   REGION Sequence Next Step Condition
       IF #sCheck_Step_Condition THEN
           CASE #sCurrent_Step_NB OF
               #S00_INIT:
                   REGION S00 INIT
                       IF #sInterface.SequenceReleased AND #iJobReq THEN
                           #sCurrent_Step_NB := #S10_CHECK_INT_LOAD_UNLOAD_OPTION;
                           #sInterface.SequenceRun := TRUE;
                           #sCheck_Step_Condition := FALSE;
                       ELSE
                           #sInterface.SequenceRun := FALSE;
                       END_IF;
                   END_REGION
               #S10_CHECK_INT_LOAD_UNLOAD_OPTION:
                   REGION S10_CHECK_INT_LOAD_UNLOAD_OPTION
                       IF #sInterface.SequenceReleased AND #sStepForward AND "DB_LoaderOptions".IntLoadUnload.CommonPos AND (#iDrilledPartToUnload OR #iUnDrilledPartToLoad) THEN
                           #sCurrent_Step_NB := #S20_SHUTTLE_TO_INT_LOAD_UNLOAD_POS_START_REQ;
                           #sCheck_Step_Condition := FALSE;
                       ELSIF #sInterface.SequenceReleased AND #sStepForward AND "DB_LoaderOptions".IntLoadUnload.CommonPos AND NOT #iJobReq OR (NOT #iDrilledPartToUnload AND NOT #iUnDrilledPartToLoad) THEN
                           #sCurrent_Step_NB := #S260_NO_PART_TO_LOAD_UNLOAD;
                           #sCheck_Step_Condition := FALSE;
                       END_IF;
                   END_REGION
               #S20_SHUTTLE_TO_INT_LOAD_UNLOAD_POS_START_REQ:
                   REGION S20_SHUTTLE_TO_INT_LOAD_UNLOAD_POS_START_REQ
                       IF #sInterface.SequenceReleased AND (#iShuttleMoving OR #iShuttleIntLoadUnloadPos) THEN
                           #sCurrent_Step_NB := #S30_SHUTTLE_TO_INT_LOAD_UNLOAD_POS_REACHED;
                           #sCheck_Step_Condition := FALSE;
                       END_IF;
                   END_REGION
               #S30_SHUTTLE_TO_INT_LOAD_UNLOAD_POS_REACHED:
                   REGION S30_SHUTTLE_TO_INT_LOAD_UNLOAD_POS_REACHED
                       IF #sInterface.SequenceReleased AND #sStepForward AND NOT #sShuttleStartReq AND #iShuttleIntLoadUnloadPos THEN
                           #sCurrent_Step_NB := #S60_AXIS_V_TO_INT_LOAD_UNLOAD_POS_START_REQ;
                           #sCheck_Step_Condition := FALSE;
                       END_IF;
                   END_REGION
               #S40_AXIS_W_TO_SAFE_POS_START_REQ:
                   REGION S40_AXIS_W_TO_SAFE_POS_START_REQ
                       IF #sInterface.SequenceReleased AND #sStepForward AND (#iAxisW_Moving OR #iAxisW_SafePos) THEN
                           #sCurrent_Step_NB := #S50_AXIS_W_TO_SAFE_POS_REACHED;
                           #sCheck_Step_Condition := FALSE;
                       END_IF;
                   END_REGION
               #S50_AXIS_W_TO_SAFE_POS_REACHED:
                   REGION S50_AXIS_W_TO_SAFE_POS_REACHED
                       IF #sInterface.SequenceReleased AND #sStepForward AND NOT #sAxisW_StartReq AND #iAxisW_SafePos THEN
                           #sCurrent_Step_NB := #S60_AXIS_V_TO_INT_LOAD_UNLOAD_POS_START_REQ;
                           #sCheck_Step_Condition := FALSE;
                       END_IF;
                   END_REGION
               #S60_AXIS_V_TO_INT_LOAD_UNLOAD_POS_START_REQ:
                   REGION S60_AXIS_V_TO_INT_LOAD_UNLOAD_POS_START_REQ
                       IF #sInterface.SequenceReleased AND (#iAxisV_Moving OR #iAxisV_LoadUnloadShuttlePos) THEN
                           #sCurrent_Step_NB := #S70_AXIS_V_TO_INT_LOAD_UNLOAD_POS_REACHED;
                           #sCheck_Step_Condition := FALSE;
                       END_IF;
                   END_REGION
               #S70_AXIS_V_TO_INT_LOAD_UNLOAD_POS_REACHED:
                   REGION S70_AXIS_V_TO_INT_LOAD_UNLOAD_POS_REACHED
                       IF #sInterface.SequenceReleased AND #sStepForward AND NOT #sAxisV_StartReq AND #iAxisV_LoadUnloadShuttlePos THEN
                           #sCurrent_Step_NB := #S80_AXIS_W_TO_INT_LOAD_UNLOAD_APPROACH_POS_START_REQ;
                           #sCheck_Step_Condition := FALSE;
                       END_IF;
                   END_REGION
               #S80_AXIS_W_TO_INT_LOAD_UNLOAD_APPROACH_POS_START_REQ:
                   REGION S80_AXIS_W_TO_INT_LOAD_UNLOAD_APPROACH_POS_START_REQ
                       IF #sInterface.SequenceReleased AND (#iAxisW_Moving OR #iAxisW_ApproachLoadUnloadPos) THEN
                           #sCurrent_Step_NB := #S90_AXIS_W_TO_INT_LOAD_UNLOAD_APPROACH_POS_REACHED;
                           #sCheck_Step_Condition := FALSE;
                       END_IF;
                   END_REGION
               #S90_AXIS_W_TO_INT_LOAD_UNLOAD_APPROACH_POS_REACHED:
                   REGION S90_AXIS_W_TO_INT_LOAD_UNLOAD_APPROACH_POS_REACHED
                       IF #sInterface.SequenceReleased AND #sStepForward AND NOT #sAxisW_StartReq AND #iAxisW_ApproachLoadUnloadPos THEN
                           #sCurrent_Step_NB := #S100_AXIS_W_TO_INT_LOAD_UNLOAD_POS_START_REQ;
                           #sCheck_Step_Condition := FALSE;
                       END_IF;
                   END_REGION
               #S100_AXIS_W_TO_INT_LOAD_UNLOAD_POS_START_REQ:
                   REGION S100_AXIS_W_TO_INT_LOAD_UNLOAD_POS_START_REQ
                       IF #sInterface.SequenceReleased AND (#iAxisW_Moving OR #iAxisW_LoadUnloadPos) THEN
                           #sCurrent_Step_NB := #S110_AXIS_W_TO_INT_LOAD_UNLOAD_POS_REACHED;
                           #sCheck_Step_Condition := FALSE;
                       END_IF;
                   END_REGION
               #S110_AXIS_W_TO_INT_LOAD_UNLOAD_POS_REACHED:
                   REGION S110_AXIS_W_TO_INT_LOAD_UNLOAD_POS_REACHED
                       IF #sInterface.SequenceReleased AND #sStepForward AND NOT #sAxisW_StartReq AND #iAxisW_LoadUnloadPos THEN
                           #sCurrent_Step_NB := #S120_CLOSE_LOAD_GRIPPER;
                           #sCheck_Step_Condition := FALSE;
                       END_IF;
                   END_REGION
               #S120_CLOSE_LOAD_GRIPPER:
                   REGION S120_CLOSE_LOAD_GRIPPER
                       IF #sInterface.SequenceReleased AND #sStepForward
                           AND ((#iUnDrilledPartToLoad AND #iLoadGripperClosed) OR NOT #iUnDrilledPartToLoad) THEN
                           #sCurrent_Step_NB := #S130_AXIS_W_TO_SAFE_POS_START_REQ;
                           #sCheck_Step_Condition := FALSE;
                       END_IF;
                   END_REGION
               #S130_AXIS_W_TO_SAFE_POS_START_REQ:
                   REGION S130_AXIS_W_TO_SAFE_POS_START_REQ
                       IF #sInterface.SequenceReleased AND (#iAxisW_Moving OR #iAxisW_SafePos) THEN
                           #sCurrent_Step_NB := #S140_AXIS_W_TO_SAFE_POS_REACHED;
                           #sCheck_Step_Condition := FALSE;
                       END_IF;
                   END_REGION
               #S140_AXIS_W_TO_SAFE_POS_REACHED:
                   REGION S140_AXIS_W_TO_SAFE_POS_REACHED
                       IF #sInterface.SequenceReleased AND #sStepForward AND NOT #sAxisW_StartReq AND #iAxisW_SafePos THEN
                           #sCurrent_Step_NB := #S150_SHUTTLE_TO_INT_LOAD_UNLOAD_OP_POS_START_REQ;
                           #sCheck_Step_Condition := FALSE;
                       END_IF;
                   END_REGION
               #S150_SHUTTLE_TO_INT_LOAD_UNLOAD_OP_POS_START_REQ:
                   REGION S150_SHUTTLE_TO_INT_LOAD_UNLOAD_OP_POS_START_REQ
                       IF #sInterface.SequenceReleased AND (#iShuttleMoving OR #iShuttleIntLoadUnloadOP_Pos) THEN
                           #sCurrent_Step_NB := #S160_SHUTTLE_TO_INT_LOAD_UNLOAD_OP_POS_REACHED;
                           #sCheck_Step_Condition := FALSE;
                       END_IF;
                   END_REGION
               #S160_SHUTTLE_TO_INT_LOAD_UNLOAD_OP_POS_REACHED:
                   REGION S160_SHUTTLE_TO_INT_LOAD_UNLOAD_OP_POS_REACHED
                       IF #sInterface.SequenceReleased AND #sStepForward AND NOT #sShuttleStartReq AND #iShuttleIntLoadUnloadOP_Pos THEN
                           #sCurrent_Step_NB := #S170_AXIS_W_TO_INT_LOAD_UNLOAD_APPROACH_POS_START_REQ;
                           #sCheck_Step_Condition := FALSE;
                       END_IF;
                   END_REGION
               #S170_AXIS_W_TO_INT_LOAD_UNLOAD_APPROACH_POS_START_REQ:
                   REGION S170_AXIS_W_TO_INT_LOAD_UNLOAD_APPROACH_POS_START_REQ
                       IF #sInterface.SequenceReleased AND (#iAxisW_Moving OR #iAxisW_ApproachLoadUnloadPos) THEN
                           #sCurrent_Step_NB := #S180_AXIS_W_TO_INT_LOAD_UNLOAD_APPROACH_POS_REACHED;
                           #sCheck_Step_Condition := FALSE;
                       END_IF;
                   END_REGION
               #S180_AXIS_W_TO_INT_LOAD_UNLOAD_APPROACH_POS_REACHED:
                   REGION S180_AXIS_W_TO_INT_LOAD_UNLOAD_APPROACH_POS_REACHED
                       IF #sInterface.SequenceReleased AND #sStepForward AND NOT #sAxisW_StartReq AND #iAxisW_ApproachLoadUnloadPos THEN
                           #sCurrent_Step_NB := #S190_AXIS_W_TO_INT_LOAD_UNLOAD_POS_START_REQ;
                           #sCheck_Step_Condition := FALSE;
                       END_IF;
                   END_REGION
               #S190_AXIS_W_TO_INT_LOAD_UNLOAD_POS_START_REQ:
                   REGION S190_AXIS_W_TO_INT_LOAD_UNLOAD_POS_START_REQ
                       IF #sInterface.SequenceReleased AND (#iAxisW_Moving OR #iAxisW_LoadUnloadPos) THEN
                           #sCurrent_Step_NB := #S200_AXIS_W_TO_INT_LOAD_UNLOAD_POS_REACHED;
                           #sCheck_Step_Condition := FALSE;
                       END_IF;
                   END_REGION
               #S200_AXIS_W_TO_INT_LOAD_UNLOAD_POS_REACHED:
                   REGION S200_AXIS_W_TO_INT_LOAD_UNLOAD_POS_REACHED
                       IF #sInterface.SequenceReleased AND #sStepForward AND NOT #sAxisW_StartReq AND #iAxisW_LoadUnloadPos THEN
                           #sCurrent_Step_NB := #S210_OPEN_UNLOAD_GRIPPER;
                           #sCheck_Step_Condition := FALSE;
                       END_IF;
                   END_REGION
               #S210_OPEN_UNLOAD_GRIPPER:
                   REGION S210_OPEN_UNLOAD_GRIPPER
                       IF #sInterface.SequenceReleased AND #sStepForward
                           AND (#iDrilledPartToUnload AND #iUnloadGripperOpen OR NOT #iDrilledPartToUnload) THEN
                           #sCurrent_Step_NB := #S220_AXIS_W_TO_SAFE_POS_START_REQ;
                           #sCheck_Step_Condition := FALSE;
                       END_IF;
                   END_REGION
               #S220_AXIS_W_TO_SAFE_POS_START_REQ:
                   REGION S220_AXIS_W_TO_SAFE_POS_START_REQ
                       IF #sInterface.SequenceReleased AND (#iAxisW_Moving OR #iAxisW_SafePos) THEN
                           #sCurrent_Step_NB := #S230_AXIS_W_TO_SAFE_POS_REACHED;
                           #sCheck_Step_Condition := FALSE;
                       END_IF;
                   END_REGION
               #S230_AXIS_W_TO_SAFE_POS_REACHED:
                   REGION S230_AXIS_W_TO_SAFE_POS_REACHED
                       IF #sInterface.SequenceReleased AND #sStepForward AND NOT #sAxisW_StartReq AND #iAxisW_SafePos THEN
                           #sCurrent_Step_NB := #S295_JOB_DONE;
                           #sCheck_Step_Condition := FALSE;
                       END_IF;
                   END_REGION
               #S240_AXIS_V_TO_SAFE_POS_START_REQ:
                   REGION S240_AXIS_V_TO_SAFE_POS_START_REQ
                       IF #sInterface.SequenceReleased AND (#iAxisV_Moving OR #iAxisV_SafePos) THEN
                           #sCurrent_Step_NB := #S250_AXIS_V_TO_SAFE_POS_REACHED;
                           #sCheck_Step_Condition := FALSE;
                       END_IF;
                   END_REGION
               #S250_AXIS_V_TO_SAFE_POS_REACHED:
                   REGION S160_AXIS_V_TO_SAFE_POS_REACHED
                       IF #sInterface.SequenceReleased AND #sStepForward AND NOT #sAxisV_StartReq AND #iAxisV_SafePos THEN
                           #sCurrent_Step_NB := #S295_JOB_DONE;
                           #sCheck_Step_Condition := FALSE;
                       END_IF;
                   END_REGION
               #S260_NO_PART_TO_LOAD_UNLOAD:
                   REGION S260_NO_PART_TO_LOAD_UNLOAD
                       IF #sInterface.SequenceReleased AND #sStepForward AND "AlwaysTRUE" THEN
                           #sCurrent_Step_NB := #S220_AXIS_W_TO_SAFE_POS_START_REQ;
                           #sCheck_Step_Condition := FALSE;
                       END_IF;
                   END_REGION
               #S295_JOB_DONE:
                   REGION S95_JOB_DONE
                       IF NOT #iJobReq THEN
                           #sCurrent_Step_NB := #S00_INIT;
                           #sCheck_Step_Condition := FALSE;
                           #sInterface.JobDone := FALSE;
                       END_IF;
                   END_REGION
               ELSE
                   #sInterface.Error := TRUE;
           END_CASE;
       END_IF;
   END_REGION

   REGION Outputs Update
       #oShuttleStartReq := #sShuttleStartReq;
       #oShuttlePosSetPoint := #sShuttlePosSetPoint;
       #oAxisV_StartReq := #sAxisV_StartReq;
       #oAxisV_PosSetPoint := #sAxisV_PosSetPoint;
       #oAxisW_StartReq := #sAxisW_StartReq;
       #oAxisW_PosSetPoint := #sAxisW_PosSetPoint;
       #oLoadGripperCloseReq := #sLoadGripperCloseReq;
       #oUnloadGripperOpenReq := #sUnloadGripperOpenReq;

   END_REGION

   REGION Steps - Date and Time History
       IF #sHistory.Activation THEN
           IF #sHistory.Steps[0] <> #sCurrent_Step_NB THEN
               FOR #tIndex := 98 TO 0 BY -1 DO
                   #sHistory.Steps[#tIndex + 1] := #sHistory.Steps[#tIndex];
                   #sHistory.Date_Time[#tIndex + 1] := #sHistory.Date_Time[#tIndex];
               END_FOR;
               #sHistory.Steps[0] := #sCurrent_Step_NB;
               #sHistory.Date_Time[0] := #iPLC_DateAndTime;
           END_IF;
       END_IF;
   END_REGION

   REGION Steps Text
       #StepText(iErrorCode := #sCurrent_Step_NB,
                 oErrorText => #StepText.oErrorText);
   END_REGION
END_FUNCTION_BLOCK

FUNCTION_BLOCK "FB_PartControl"   // FB58, SCL
{ S7_Optimized_Access := 'TRUE' }
// stored: MemoryReserve 100, SetENOAutomatically false
   VAR_INPUT
      iStartSeqCond : Bool;   // Start Sequence Conditions
      iJobReq : Bool;   // Job Request - From Main
      iCtrlEnabled : Bool;   // Part Control Enable - Param or Condition
      iShuttleCtrlUndrilledPos : Bool;   // Undrilled Pos. Reached (Option Individual Ctrl) - Param
      iShuttleCtrlUndrilledPosSetPoint : LReal;   // Undrilled Pos. Setpoint (Option Individual Ctrl) - Param
      iShuttleCtrlDrilledPos : Bool;   // Drilled Pos. Reached (Option Individual Ctrl) - Param
      iShuttleCtrlDrilledPosSetPoint : LReal;   // Drilled Pos. Setpoint (Option Individual Ctrl) - Param
      iShuttleCtrlPos : Bool;   // Control Pos. Reached (Option Common Ctrl) - Param
      iShuttleCtrlPosSetPoint : LReal;   // Control Pos. Setpoint (Option Common Ctrl) - Param
      iExpectedCtrlUndrilled : Bool;   // Expected result Undrilled Pos.
      iExpectedCtrlDrilled : Bool;   // Expected result Drilled Pos.
      iPartMeasureValue : Real;   // Part Measure Value (Option Analog Measure) - From AI
      iPartMeasureTolMin : Real;   // Part Tol Min Value (Option Analog Measure) - Param
      iPartMeasureTolMax : Real;   // Part Tol Max Value (Option Analog Measure) - Param
      iUndrilledPartPresence : Bool;
      iDrilledPartPresence : Bool;
      iShuttleMoving : Bool;   // Shuttle is moving - From FB_LoaderAxis
      iShuttleInPos : Bool;   // Shuttle pos. reached - From FB_LoaderAxis
      iPLC_DateAndTime : DTL;
      iStepPause : Bool;
   END_VAR
   VAR_OUTPUT
      oShuttleStartReq { ExternalAccessible := 'False'; ExternalVisible := 'False'; ExternalWritable := 'False'} : Bool;   // Shuttle Start Order - To FB_LoaderAxis
      oShuttlePosSetPoint { ExternalAccessible := 'False'; ExternalVisible := 'False'; ExternalWritable := 'False'} : Real;   // Shuttle Position Setpoint - To FB_LoaderAxis
      oPartControlOK : Bool;   // Part OK - To Main
      oPartControlNOK : Bool;   // Part NOK - To Main
   END_VAR
   VAR
      sCurrent_Step_NB : Int;   // Active Step Number
      sCheck_Step_Condition : Bool;
      sOneStepForward : Bool;
      sRTOneStepForward : R_TRIG;
      sOneStepMode { S7_SetPoint := 'True'} : Bool;
      sStepForward : Bool;
      sInterface : "UDT_SequenceInterface";
      sShuttleStartReq { ExternalAccessible := 'False'; ExternalVisible := 'False'; ExternalWritable := 'False'} : Bool;
      sShuttlePosSetPoint { ExternalAccessible := 'False'; ExternalVisible := 'False'; ExternalWritable := 'False'} : Real;
      sMissingPartCtrlUndrilled : Bool;
      sMissingPartCtrlDrilled : Bool;
      sExtraPartCtrlUndrilled : Bool;
      sExtraPartCtrlDrilled : Bool;
      sPresencePartUndrilledPos : Bool;
      sPresencePartDrilledPos : Bool;
      sPartControlOK : Bool;
      sPartControlNOK : Bool;
      sControlTimer : TON_TIME;
      sHistory : Struct
         Activation : Bool;
         Steps : Array[0..99] of Int;
         Date_Time : Array[0..99] of DTL;
      END_STRUCT;
      StepText : "FB_GetTextErrorCode";
   END_VAR
   VAR_TEMP
      tIndex : Int;   // Index
   END_VAR
   VAR CONSTANT
      S00_INIT : Int := 0;
      S10_CHECK_PART_PRESENCE_OPTION : Int := 10;
      S20_SHUTTLE_TO_UNDRILLED_POS_START_REQ : Int := 20;
      S30_SHUTTLE_TO_UNDRILLED_POS_REACHED : Int := 30;
      S40_WAIT_UNDRILLED_CTRL_EXECUTION : Int := 40;
      S50_SHUTTLE_TO_DRILLED_POS_START_REQ : Int := 50;
      S60_SHUTTLE_TO_DRILLED_POS_REACHED : Int := 60;
      S70_WAIT_DRILLED_CTRL_EXECUTION : Int := 70;
      S80_CHECK_PART_POS_RESULT : Int := 80;
      S120_SHUTTLE_TO_CONTROL_POS_START_REQ : Int := 120;
      S130_SHUTTLE_TO_CONTROL_POS_REACHED : Int := 130;
      S140_WAIT_CONTROL_EXECUTION : Int := 140;
      S180_CHECK_PART_POS_RESULT : Int := 180;
      S280_NO_PART_CTRL : Int := 280;
      S295_JOB_DONE : Int := 295;
   END_VAR
   // StepText.sCode_error[0].ErrorCode := 0;
   // StepText.sCode_error[1].ErrorCode := 10;
   // StepText.sCode_error[2].ErrorCode := 20;
   // StepText.sCode_error[3].ErrorCode := 30;
   // StepText.sCode_error[4].ErrorCode := 40;
   // StepText.sCode_error[5].ErrorCode := 50;
   // StepText.sCode_error[6].ErrorCode := 60;
   // StepText.sCode_error[7].ErrorCode := 70;
   // StepText.sCode_error[8].ErrorCode := 80;
   // StepText.sCode_error[9].ErrorCode := 90;
   // StepText.sCode_error[10].ErrorCode := 95;
BEGIN
   REGION Description header 
       //==================================================================================
       // POSALUX Swiss SA / (C) Copyright 2025
       //----------------------------------------------------------------------------------
       // Title: FB_PartControl
       // Comment/Function: 
       // Author: Fabien WALDT
       // Engineering: TIA Portal v17
       //----------------------------------------------------------------------------------
       // Change log table:
       // Version  | Date     | Expert in charge | Changes applied
       // ---------|----------|------------------|-----------------------------------------
       // 00.00.01 | 20250527 | WFA              | First released version
       // =================================================================================
   END_REGION

   REGION Define condition to start
       IF #iStartSeqCond THEN
           #sInterface.SequenceReleased := TRUE;
       ELSE
           // Standard sequencer controls
           #sInterface.SequenceReleased := FALSE;
           #sCurrent_Step_NB := #S00_INIT;
           #sInterface.SequenceRun := FALSE;
           #sInterface.JobDone := FALSE;
           #sCheck_Step_Condition := FALSE;

           // Dedicated sequencer controls
           #sShuttleStartReq := FALSE;
           #sShuttlePosSetPoint := 0.0;
           #sPresencePartUndrilledPos := FALSE;
           #sPresencePartDrilledPos := FALSE;

           // Add specifics controls 
       END_IF;

       // Reset interface error
       IF #sInterface.Reset THEN
           #sInterface.Error := FALSE;
       END_IF;

       // Reset start when axis in position
       IF #iShuttleInPos THEN
           #sShuttleStartReq := FALSE;
       END_IF;

       // One step forward
       #sRTOneStepForward.CLK := #sOneStepForward;
       #sRTOneStepForward();
       #sStepForward := (NOT #sOneStepMode OR (#sOneStepMode AND #sRTOneStepForward.Q)) AND NOT #iStepPause;
       #sOneStepForward := FALSE;

       // Step Timer
       #sControlTimer(IN := #sCurrent_Step_NB = 40 OR #sCurrent_Step_NB = 140,
                            PT := T#50ms);
   END_REGION

   REGION Sequence Function
       CASE #sCurrent_Step_NB OF
           #S00_INIT:
               REGION S00 INIT
                   #sCheck_Step_Condition := TRUE;
               END_REGION
           #S10_CHECK_PART_PRESENCE_OPTION:
               REGION S10_CHECK_PART_PRESENCE_OPTION
                   #sPartControlOK := FALSE;
                   #sPartControlNOK := FALSE;
                   #sMissingPartCtrlUndrilled := FALSE;
                   #sMissingPartCtrlDrilled := FALSE;
                   #sExtraPartCtrlUndrilled := FALSE;
                   #sExtraPartCtrlDrilled := FALSE;
                   #sCheck_Step_Condition := TRUE;
               END_REGION
           #S20_SHUTTLE_TO_UNDRILLED_POS_START_REQ:
               REGION S20_SHUTTLE_TO_UNDRILLED_POS_START_REQ
                   #sShuttleStartReq := NOT #iShuttleCtrlUndrilledPos;
                   #sShuttlePosSetPoint := LREAL_TO_REAL(#iShuttleCtrlUndrilledPosSetPoint);
                   #sCheck_Step_Condition := TRUE;
               END_REGION
           #S30_SHUTTLE_TO_UNDRILLED_POS_REACHED:
               REGION S30_SHUTTLE_TO_UNDRILLED_POS_REACHED
                   #sCheck_Step_Condition := TRUE;
               END_REGION
           #S40_WAIT_UNDRILLED_CTRL_EXECUTION:
               REGION S40_WAIT_UNDRILLED_CTRL_EXECUTION
                   IF "DB_LoaderOptions".PartControl.AnalogMeasure THEN
                       IF #iPartMeasureValue > #iPartMeasureTolMin AND #iPartMeasureValue < #iPartMeasureTolMax THEN
                           #sPresencePartUndrilledPos := TRUE;
                       ELSE
                           #sPresencePartUndrilledPos := FALSE;
                       END_IF;
                   ELSIF "DB_LoaderOptions".PartControl.DigitalMeasure THEN
                       IF #iUndrilledPartPresence THEN
                           #sPresencePartUndrilledPos := TRUE;
                       ELSE
                           #sPresencePartUndrilledPos := FALSE;
                       END_IF;
                       IF #iDrilledPartPresence THEN
                           #sPresencePartDrilledPos := TRUE;
                       ELSE
                           #sPresencePartDrilledPos := FALSE;
                       END_IF;
                   ELSE
                       #sInterface.Error := TRUE;
                   END_IF;
                   IF #sControlTimer.Q THEN
                       #sCheck_Step_Condition := TRUE;
                   END_IF;
               END_REGION
           #S50_SHUTTLE_TO_DRILLED_POS_START_REQ:
               REGION S50_SHUTTLE_TO_DRILLED_POS_START_REQ
                   #sShuttleStartReq := NOT #iShuttleCtrlDrilledPos;
                   #sShuttlePosSetPoint := LREAL_TO_REAL(#iShuttleCtrlDrilledPosSetPoint);
                   #sCheck_Step_Condition := TRUE;
               END_REGION
           #S60_SHUTTLE_TO_DRILLED_POS_REACHED:
               REGION S60_SHUTTLE_TO_DRILLED_POS_REACHED
                   #sCheck_Step_Condition := TRUE;
               END_REGION
           #S70_WAIT_DRILLED_CTRL_EXECUTION:
               REGION S70_WAIT_DRILLED_CTRL_EXECUTION
                   IF "DB_LoaderOptions".PartControl.AnalogMeasure THEN
                       IF #iPartMeasureValue > #iPartMeasureTolMin AND #iPartMeasureValue < #iPartMeasureTolMax THEN
                           #sPresencePartUndrilledPos := TRUE;
                       ELSE
                           #sPresencePartUndrilledPos := FALSE;
                       END_IF;
                   ELSIF "DB_LoaderOptions".PartControl.DigitalMeasure THEN
                       IF #iUndrilledPartPresence THEN
                           #sPresencePartUndrilledPos := TRUE;
                       ELSE
                           #sPresencePartUndrilledPos := FALSE;
                       END_IF;
                   ELSE
                       #sInterface.Error := TRUE;
                   END_IF;
                   #sCheck_Step_Condition := TRUE;
               END_REGION
           #S80_CHECK_PART_POS_RESULT:
               REGION S80_CHECK_PART_POS_RESULT
                   #sExtraPartCtrlUndrilled := #sPresencePartUndrilledPos AND NOT #iExpectedCtrlUndrilled;
                   #sMissingPartCtrlUndrilled := NOT #sPresencePartUndrilledPos AND #iExpectedCtrlUndrilled;
                   #sExtraPartCtrlDrilled := #sPresencePartDrilledPos AND NOT #iExpectedCtrlDrilled;
                   #sMissingPartCtrlDrilled := NOT #sPresencePartDrilledPos AND #iExpectedCtrlDrilled;

                   IF #sPresencePartUndrilledPos = #iExpectedCtrlUndrilled AND #sPresencePartDrilledPos = #iExpectedCtrlDrilled THEN
                       #sPartControlOK := TRUE;
                       #sPartControlNOK := FALSE;
                   ELSE
                       #sPartControlOK := FALSE;
                       #sPartControlNOK := TRUE;
                   END_IF;
                   #sCheck_Step_Condition := TRUE;
               END_REGION

           #S120_SHUTTLE_TO_CONTROL_POS_START_REQ:
               REGION S120_SHUTTLE_TO_CONTROL_POS_START_REQ
                   #sShuttleStartReq := NOT #iShuttleCtrlPos;
                   #sShuttlePosSetPoint := LREAL_TO_REAL(#iShuttleCtrlPosSetPoint);
                   #sCheck_Step_Condition := TRUE;
               END_REGION
           #S130_SHUTTLE_TO_CONTROL_POS_REACHED:
               REGION S130_SHUTTLE_TO_CONTROL_POS_REACHED
                   #sCheck_Step_Condition := TRUE;
               END_REGION
           #S140_WAIT_CONTROL_EXECUTION:
               REGION S140_WAIT_CONTROL_EXECUTION
                   IF "DB_LoaderOptions".PartControl.AnalogMeasure THEN
                       IF #iPartMeasureValue > #iPartMeasureTolMin AND #iPartMeasureValue < #iPartMeasureTolMax THEN
                           #sPresencePartUndrilledPos := TRUE;
                       ELSE
                           #sPresencePartUndrilledPos := FALSE;
                       END_IF;
                   ELSIF "DB_LoaderOptions".PartControl.DigitalMeasure THEN
                       IF #iUndrilledPartPresence THEN
                           #sPresencePartUndrilledPos := TRUE;
                       ELSE
                           #sPresencePartUndrilledPos := FALSE;
                       END_IF;
                       IF #iDrilledPartPresence THEN
                           #sPresencePartDrilledPos := TRUE;
                       ELSE
                           #sPresencePartDrilledPos := FALSE;
                       END_IF;
                   ELSE
                       #sInterface.Error := TRUE;
                   END_IF;
                   IF #sControlTimer.Q THEN
                       #sCheck_Step_Condition := TRUE;
                   END_IF;
               END_REGION
           #S180_CHECK_PART_POS_RESULT:
               REGION S180_CHECK_PART_POS_RESULT
                   #sExtraPartCtrlUndrilled := #sPresencePartUndrilledPos AND NOT #iExpectedCtrlUndrilled;
                   #sMissingPartCtrlUndrilled := NOT #sPresencePartUndrilledPos AND #iExpectedCtrlUndrilled;
                   #sExtraPartCtrlDrilled := #sPresencePartDrilledPos AND NOT #iExpectedCtrlDrilled;
                   #sMissingPartCtrlDrilled := NOT #sPresencePartDrilledPos AND #iExpectedCtrlDrilled;

                   IF #sPresencePartUndrilledPos = #iExpectedCtrlUndrilled AND #sPresencePartDrilledPos = #iExpectedCtrlDrilled THEN
                       #sPartControlOK := TRUE;
                       #sPartControlNOK := FALSE;
                   ELSE
                       #sPartControlOK := FALSE;
                       #sPartControlNOK := TRUE;
                   END_IF;
                   #sCheck_Step_Condition := TRUE;
               END_REGION

           #S280_NO_PART_CTRL:
               REGION S280_NO_PART_CTRL
                   #sPartControlOK := TRUE;
                   #sPartControlNOK := FALSE;
                   #sCheck_Step_Condition := TRUE;
               END_REGION

           #S295_JOB_DONE:
               REGION S295_JOB_DONE
                   #sInterface.JobDone := TRUE;
                   #sCheck_Step_Condition := TRUE;
               END_REGION
           ELSE:
               #sInterface.Error := TRUE;
       END_CASE;
   END_REGION

   REGION Sequence Next Step Condition
       IF #sCheck_Step_Condition THEN
           CASE #sCurrent_Step_NB OF
               #S00_INIT:
                   REGION S00 INIT
                       IF #sInterface.SequenceReleased AND #iJobReq THEN
                           #sCurrent_Step_NB := #S10_CHECK_PART_PRESENCE_OPTION;
                           #sInterface.SequenceRun := TRUE;
                           #sCheck_Step_Condition := FALSE;
                       ELSE
                           #sInterface.SequenceRun := FALSE;
                       END_IF;
                   END_REGION
               #S10_CHECK_PART_PRESENCE_OPTION:
                   REGION S10_CHECK_PART_PRESENCE_OPTION
                       IF #sInterface.SequenceReleased AND #sStepForward AND "DB_LoaderOptions".PartControl.Individual AND (NOT "DB_LoaderOptions".PartControl.Disabled AND #iCtrlEnabled) THEN
                           #sCurrent_Step_NB := #S20_SHUTTLE_TO_UNDRILLED_POS_START_REQ;
                           #sCheck_Step_Condition := FALSE;
                       ELSIF #sInterface.SequenceReleased AND #sStepForward AND "DB_LoaderOptions".PartControl.Common AND (NOT "DB_LoaderOptions".PartControl.Disabled AND #iCtrlEnabled) THEN
                           #sCurrent_Step_NB := #S120_SHUTTLE_TO_CONTROL_POS_START_REQ;
                           #sCheck_Step_Condition := FALSE;
                       ELSIF #sInterface.SequenceReleased AND #sStepForward AND ("DB_LoaderOptions".PartControl.Disabled OR NOT #iCtrlEnabled) THEN
                           #sCurrent_Step_NB := #S280_NO_PART_CTRL;
                           #sCheck_Step_Condition := FALSE;
                       END_IF;
                   END_REGION
               #S20_SHUTTLE_TO_UNDRILLED_POS_START_REQ:
                   REGION S20_SHUTTLE_TO_UNDRILLED_POS_START_REQ
                       IF #sInterface.SequenceReleased AND (#iShuttleMoving OR #iShuttleCtrlUndrilledPos) THEN
                           #sCurrent_Step_NB := #S30_SHUTTLE_TO_UNDRILLED_POS_REACHED;
                           #sCheck_Step_Condition := FALSE;
                       END_IF;
                   END_REGION
               #S30_SHUTTLE_TO_UNDRILLED_POS_REACHED:
                   REGION S30_SHUTTLE_TO_UNDRILLED_POS_REACHED
                       IF #sInterface.SequenceReleased AND #sStepForward AND NOT #sShuttleStartReq AND #iShuttleCtrlUndrilledPos THEN
                           #sCurrent_Step_NB := #S40_WAIT_UNDRILLED_CTRL_EXECUTION;
                           #sCheck_Step_Condition := FALSE;
                       END_IF;
                   END_REGION
               #S40_WAIT_UNDRILLED_CTRL_EXECUTION:
                   REGION S40_WAIT_UNDRILLED_CTRL_EXECUTION
                       IF #sInterface.SequenceReleased AND #sStepForward AND "AlwaysTRUE" THEN
                           #sCurrent_Step_NB := #S50_SHUTTLE_TO_DRILLED_POS_START_REQ;
                           #sCheck_Step_Condition := FALSE;
                       END_IF;
                   END_REGION
               #S50_SHUTTLE_TO_DRILLED_POS_START_REQ:
                   REGION S50_SHUTTLE_TO_DRILLED_POS_START_REQ
                       IF #sInterface.SequenceReleased AND (#iShuttleMoving OR #iShuttleCtrlDrilledPos) THEN
                           #sCurrent_Step_NB := #S60_SHUTTLE_TO_DRILLED_POS_REACHED;
                           #sCheck_Step_Condition := FALSE;
                       END_IF;
                   END_REGION
               #S60_SHUTTLE_TO_DRILLED_POS_REACHED:
                   REGION S60_SHUTTLE_TO_DRILLED_POS_REACHED
                       IF #sInterface.SequenceReleased AND #sStepForward AND NOT #sShuttleStartReq AND #iShuttleCtrlDrilledPos THEN
                           #sCurrent_Step_NB := #S70_WAIT_DRILLED_CTRL_EXECUTION;
                           #sCheck_Step_Condition := FALSE;
                       END_IF;
                   END_REGION
               #S70_WAIT_DRILLED_CTRL_EXECUTION:
                   REGION S70_WAIT_DRILLED_CTRL_EXECUTION
                       IF #sInterface.SequenceReleased AND #sStepForward AND "AlwaysTRUE" THEN
                           #sCurrent_Step_NB := #S80_CHECK_PART_POS_RESULT;
                           #sCheck_Step_Condition := FALSE;
                       END_IF;
                   END_REGION
               #S80_CHECK_PART_POS_RESULT:
                   REGION S80_CHECK_PART_POS_RESULT
                       IF #sInterface.SequenceReleased AND #sStepForward AND "AlwaysTRUE" THEN
                           #sCurrent_Step_NB := #S295_JOB_DONE;
                           #sCheck_Step_Condition := FALSE;
                       END_IF;
                   END_REGION

               #S120_SHUTTLE_TO_CONTROL_POS_START_REQ:
                   REGION S120_SHUTTLE_TO_CONTROL_POS_START_REQ
                       IF #sInterface.SequenceReleased AND (#iShuttleMoving OR #iShuttleCtrlPos) THEN
                           #sCurrent_Step_NB := #S130_SHUTTLE_TO_CONTROL_POS_REACHED;
                           #sCheck_Step_Condition := FALSE;
                       END_IF;
                   END_REGION
               #S130_SHUTTLE_TO_CONTROL_POS_REACHED:
                   REGION S130_SHUTTLE_TO_CONTROL_POS_REACHED
                       IF #sInterface.SequenceReleased AND #sStepForward AND NOT #sShuttleStartReq AND #iShuttleCtrlPos THEN
                           #sCurrent_Step_NB := #S140_WAIT_CONTROL_EXECUTION;
                           #sCheck_Step_Condition := FALSE;
                       END_IF;
                   END_REGION
               #S140_WAIT_CONTROL_EXECUTION:
                   REGION S140_WAIT_CONTROL_EXECUTION
                       IF #sInterface.SequenceReleased AND #sStepForward AND "AlwaysTRUE" THEN
                           #sCurrent_Step_NB := #S180_CHECK_PART_POS_RESULT;
                           #sCheck_Step_Condition := FALSE;
                       END_IF;
                   END_REGION
               #S180_CHECK_PART_POS_RESULT:
                   REGION S180_CHECK_PART_POS_RESULT
                       IF #sInterface.SequenceReleased AND #sStepForward AND "AlwaysTRUE" THEN
                           #sCurrent_Step_NB := #S295_JOB_DONE;
                           #sCheck_Step_Condition := FALSE;
                       END_IF;
                   END_REGION

               #S280_NO_PART_CTRL:
                   REGION S280_NO_PART_CTRL
                       IF #sInterface.SequenceReleased AND #sStepForward AND "AlwaysTRUE" THEN
                           #sCurrent_Step_NB := #S295_JOB_DONE;
                           #sCheck_Step_Condition := FALSE;
                       END_IF;
                   END_REGION

               #S295_JOB_DONE:
                   REGION S95_JOB_DONE
                       IF NOT #iJobReq THEN
                           #sCurrent_Step_NB := #S00_INIT;
                           #sCheck_Step_Condition := FALSE;
                           #sInterface.JobDone := FALSE;
                       END_IF;
                   END_REGION
               ELSE
                   #sInterface.Error := TRUE;
           END_CASE;
       END_IF;
   END_REGION

   REGION Outputs Update
       #oShuttleStartReq := #sShuttleStartReq;
       #oShuttlePosSetPoint:= #sShuttlePosSetPoint;
       #oPartControlOK := #sPartControlOK;
       #oPartControlNOK := #sPartControlNOK;
   END_REGION

   REGION Steps - Date and Time History
       IF #sHistory.Activation THEN
           IF #sHistory.Steps[0] <> #sCurrent_Step_NB THEN
               FOR #tIndex := 98 TO 0 BY -1 DO
                   #sHistory.Steps[#tIndex + 1] := #sHistory.Steps[#tIndex];
                   #sHistory.Date_Time[#tIndex + 1] := #sHistory.Date_Time[#tIndex];
               END_FOR;
               #sHistory.Steps[0] := #sCurrent_Step_NB;
               #sHistory.Date_Time[0] := #iPLC_DateAndTime;
           END_IF;
       END_IF;
   END_REGION

   REGION Steps Text
       #StepText(iErrorCode := #sCurrent_Step_NB,
                 oErrorText => #StepText.oErrorText);
   END_REGION
END_FUNCTION_BLOCK

FUNCTION_BLOCK "FB_BwLoadUnload"   // FB72, SCL
{ S7_Optimized_Access := 'TRUE' }
// stored: AutoNumber false, MemoryReserve 100, SetENOAutomatically false
   VAR_INPUT
      iStartSeqCond : Bool;   // Start Sequence Conditions
      iJobReq : Bool;   // Job Request - From Main
      iLoadReq : Bool;   // Load Request - From Main
      iUnloadReq : Bool;   // Unload Request - From Main
      iShuttleBwUnloadPos : Bool;   // Unload Pos. Reached - Param
      iShuttleBwUnloadPosSetPoint : LReal;   // Unload Pos. Setpoint - Param
      iShuttleBwLoadPos : Bool;   // Load Pos. Reached - Param
      iShuttleBwLoadPosSetPoint : LReal;   // Load Pos. Setpoint - Param
      iShuttleMoving : Bool;   // Shuttle is moving - From FB_LoaderAxis
      iShuttleInPos : Bool;   // Shuttle pos. reached - From FB_LoaderAxis
      iBwLoadDone : Bool;
      iBwUnloadDone : Bool;
      iBwLoaderInSafePos : Bool;   // Gripper in Safe Position - Param
      iPLC_DateAndTime : DTL;
      iStepPause : Bool;
   END_VAR
   VAR_OUTPUT
      oShuttleStartReq { ExternalAccessible := 'False'; ExternalVisible := 'False'; ExternalWritable := 'False'} : Bool;   // Shuttle Start Order - To FB_LoaderAxis
      oShuttlePosSetPoint { ExternalAccessible := 'False'; ExternalVisible := 'False'; ExternalWritable := 'False'} : Real;   // Shuttle Position Setpoint - To FB_LoaderAxis
      oBwLoadReq : Bool;
      oBwUnloadReq : Bool;
   END_VAR
   VAR
      sCurrent_Step_NB : Int;   // Active Step Number
      sCheck_Step_Condition : Bool;
      sOneStepForward : Bool;
      sRTOneStepForward : R_TRIG;
      sOneStepMode { S7_SetPoint := 'True'} : Bool;
      sStepForward : Bool;
      sInterface : "UDT_SequenceInterface";
      sShuttleStartReq { ExternalAccessible := 'False'; ExternalVisible := 'False'; ExternalWritable := 'False'} : Bool;
      sShuttlePosSetPoint { ExternalAccessible := 'False'; ExternalVisible := 'False'; ExternalWritable := 'False'} : Real;
      sBwLoadReq : Bool;
      sBwUnloadReq : Bool;
      sHistory : Struct
         Activation : Bool;
         Steps : Array[0..99] of Int;
         Date_Time : Array[0..99] of DTL;
      END_STRUCT;
      StepText : "FB_GetTextErrorCode";
   END_VAR
   VAR_TEMP
      tIndex : Int;   // Index
   END_VAR
   VAR CONSTANT
      S00_INIT : Int := 0;
      S10_BW_LOAD_UNLOAD_OPTION : Int := 10;
      S20_SHUTTLE_TO_BW_LOAD_POS_START_REQ : Int := 20;
      S30_SHUTTLE_TO_BW_LOAD_POS_REACHED : Int := 30;
      S40_SET_EXCHANGE_BW_LOADER_LOAD : Int := 40;
      S50_EXCHANGE_BW_LOADER_IN_PROGRESS : Int := 50;
      S60_EXCHANGE_BW_LOADER_ACQUIT : Int := 60;
      S120_SHUTTLE_TO_BW_UNLOAD_POS_START_REQ : Int := 120;
      S130_SHUTTLE_TO_BW_UNLOAD_POS_REACHED : Int := 130;
      S140_SET_EXCHANGE_BW_LOADER_UNLOAD : Int := 140;
      S150_EXCHANGE_BW_LOADER_IN_PROGRESS : Int := 150;
      S160_EXCHANGE_BW_LOADER_ACQUIT : Int := 160;
      S195_JOB_DONE : Int := 195;
   END_VAR
   // StepText.sCode_error[0].ErrorCode := 0;
   // StepText.sCode_error[1].ErrorCode := 10;
   // StepText.sCode_error[2].ErrorCode := 20;
   // StepText.sCode_error[3].ErrorCode := 30;
   // StepText.sCode_error[4].ErrorCode := 40;
   // StepText.sCode_error[5].ErrorCode := 50;
   // StepText.sCode_error[6].ErrorCode := 60;
   // StepText.sCode_error[7].ErrorCode := 70;
   // StepText.sCode_error[8].ErrorCode := 80;
   // StepText.sCode_error[9].ErrorCode := 90;
   // StepText.sCode_error[10].ErrorCode := 95;
BEGIN
   REGION Description header 
       //==================================================================================
       // POSALUX Swiss SA / (C) Copyright 2025
       //----------------------------------------------------------------------------------
       // Title: FB_BWLoadUnload
       // Comment/Function: 
       // Author: Fabien WALDT
       // Engineering: TIA Portal v17
       //----------------------------------------------------------------------------------
       // Change log table:
       // Version  | Date     | Expert in charge | Changes applied
       // ---------|----------|------------------|-----------------------------------------
       // 00.00.01 | 20250527 | WFA              | First released version
       // =================================================================================
   END_REGION

   REGION Define condition to start
       IF #iStartSeqCond THEN
           #sInterface.SequenceReleased := TRUE;
       ELSE
           // Standard sequencer controls
           #sInterface.SequenceReleased := FALSE;
           #sCurrent_Step_NB := #S00_INIT;
           #sInterface.SequenceRun := FALSE;
           #sInterface.JobDone := FALSE;
           #sCheck_Step_Condition := FALSE;

           // Dedicated sequencer controls
           #sShuttleStartReq := FALSE;
           #sShuttlePosSetPoint := 0.0;
           #sBwLoadReq := FALSE;
           #sBwUnloadReq := FALSE;
           // Add specifics controls 
       END_IF;

       // Reset interface error
       IF #sInterface.Reset THEN
           #sInterface.Error := FALSE;
       END_IF;

       // Reset start when axis in position
       IF #iShuttleInPos THEN
           #sShuttleStartReq := FALSE;
       END_IF;

       // One step forward
       #sRTOneStepForward.CLK := #sOneStepForward;
       #sRTOneStepForward();
       #sStepForward := (NOT #sOneStepMode OR (#sOneStepMode AND #sRTOneStepForward.Q)) AND NOT #iStepPause;
       #sOneStepForward := FALSE;

       // Action only true in dedicated steps

   END_REGION

   REGION Sequence Function
       CASE #sCurrent_Step_NB OF
           #S00_INIT:
               REGION S00 INIT
                   #sBwLoadReq := FALSE;
                   #sBwUnloadReq := FALSE;
                   #sCheck_Step_Condition := TRUE;
               END_REGION
           #S10_BW_LOAD_UNLOAD_OPTION:
               REGION S10_BW_LOAD_UNLOAD_OPTION

                   #sCheck_Step_Condition := TRUE;
               END_REGION
           #S20_SHUTTLE_TO_BW_LOAD_POS_START_REQ:
               REGION S20_SHUTTLE_TO_BW_LOAD_POS_START_REQ
                   #sShuttleStartReq := NOT #iShuttleBwLoadPos;
                   #sShuttlePosSetPoint := LREAL_TO_REAL(#iShuttleBwLoadPosSetPoint);
                   #sCheck_Step_Condition := TRUE;
               END_REGION
           #S30_SHUTTLE_TO_BW_LOAD_POS_REACHED:
               REGION S30_SHUTTLE_TO_BW_LOAD_POS_REACHED
                   #sCheck_Step_Condition := TRUE;
               END_REGION
           #S40_SET_EXCHANGE_BW_LOADER_LOAD:
               REGION S40_SET_EXCHANGE_BW_LOADER_LOAD
                   #sBwLoadReq := TRUE;
                   #sCheck_Step_Condition := TRUE;
               END_REGION
           #S50_EXCHANGE_BW_LOADER_IN_PROGRESS:
               REGION S50_EXCHANGE_BW_LOADER_IN_PROGRESS
                   #sCheck_Step_Condition := TRUE;
               END_REGION
           #S60_EXCHANGE_BW_LOADER_ACQUIT:
               REGION S60_EXCHANGE_BW_LOADER_ACQUIT
                   #sBwLoadReq := FALSE;
                   #sCheck_Step_Condition := TRUE;
               END_REGION

           #S120_SHUTTLE_TO_BW_UNLOAD_POS_START_REQ:
               REGION S120_SHUTTLE_TO_BW_UNLOAD_POS_START_REQ
                   #sShuttleStartReq := NOT #iShuttleBwUnloadPos;
                   #sShuttlePosSetPoint := LREAL_TO_REAL(#iShuttleBwUnloadPosSetPoint);
                   #sCheck_Step_Condition := TRUE;
               END_REGION
           #S130_SHUTTLE_TO_BW_UNLOAD_POS_REACHED:
               REGION S130_SHUTTLE_TO_BW_UNLOAD_POS_REACHED
                   #sCheck_Step_Condition := TRUE;
               END_REGION
           #S140_SET_EXCHANGE_BW_LOADER_UNLOAD:
               REGION S140_SET_EXCHANGE_BW_LOADER_UNLOAD
                   #sBwUnloadReq := TRUE;
                   #sCheck_Step_Condition := TRUE;
               END_REGION
           #S150_EXCHANGE_BW_LOADER_IN_PROGRESS:
               REGION S150_EXCHANGE_BW_LOADER_IN_PROGRESS
                   #sCheck_Step_Condition := TRUE;
               END_REGION
           #S160_EXCHANGE_BW_LOADER_ACQUIT:
               REGION S160_EXCHANGE_BW_LOADER_ACQUIT
                   #sBwUnloadReq := FALSE;
                   #sCheck_Step_Condition := TRUE;
               END_REGION
           #S195_JOB_DONE:
               REGION S95_JOB_DONE
                   #sInterface.JobDone := TRUE;
                   #sCheck_Step_Condition := TRUE;
               END_REGION
           ELSE:
               #sInterface.Error := TRUE;
       END_CASE;
   END_REGION

   REGION Sequence Next Step Condition
       IF #sCheck_Step_Condition THEN
           CASE #sCurrent_Step_NB OF
               #S00_INIT:
                   REGION S00 INIT
                       IF #sInterface.SequenceReleased AND #iJobReq THEN
                           #sCurrent_Step_NB := #S10_BW_LOAD_UNLOAD_OPTION;
                           #sInterface.SequenceRun := TRUE;
                           #sCheck_Step_Condition := FALSE;
                       ELSE
                           #sInterface.SequenceRun := FALSE;
                       END_IF;
                   END_REGION
               #S10_BW_LOAD_UNLOAD_OPTION:
                   REGION S10_BW_LOAD_UNLOAD_OPTION
                       IF #sInterface.SequenceReleased AND #sStepForward AND "DB_LoaderOptions".BwLoadUnload.SeparatePos AND #iLoadReq AND NOT #iUnloadReq THEN
                           #sCurrent_Step_NB := #S20_SHUTTLE_TO_BW_LOAD_POS_START_REQ;
                           #sCheck_Step_Condition := FALSE;
                       ELSIF #sInterface.SequenceReleased AND #sStepForward AND "DB_LoaderOptions".BwLoadUnload.SeparatePos AND NOT #iLoadReq AND #iUnloadReq THEN
                           #sCurrent_Step_NB := #S120_SHUTTLE_TO_BW_UNLOAD_POS_START_REQ;
                           #sCheck_Step_Condition := FALSE;
                       ELSIF #sInterface.SequenceReleased AND #sStepForward AND NOT #iLoadReq AND NOT #iUnloadReq THEN
                           #sCurrent_Step_NB := #S195_JOB_DONE;
                           #sCheck_Step_Condition := FALSE;
                       END_IF;
                   END_REGION
               #S20_SHUTTLE_TO_BW_LOAD_POS_START_REQ:
                   REGION S20_SHUTTLE_TO_BW_LOAD_POS_START_REQ
                       IF #sInterface.SequenceReleased AND (#iShuttleMoving OR #iShuttleBwLoadPos) THEN
                           #sCurrent_Step_NB := #S30_SHUTTLE_TO_BW_LOAD_POS_REACHED;
                           #sCheck_Step_Condition := FALSE;
                       END_IF;
                   END_REGION
               #S30_SHUTTLE_TO_BW_LOAD_POS_REACHED:
                   REGION S30_SHUTTLE_TO_BW_LOAD_POS_REACHED
                       IF #sInterface.SequenceReleased AND #sStepForward AND NOT #sShuttleStartReq AND #iShuttleBwLoadPos AND "DB_BwLoaderExchange".Inputs.BwInErrorState = 0 THEN
                           #sCurrent_Step_NB := #S40_SET_EXCHANGE_BW_LOADER_LOAD;
                           #sCheck_Step_Condition := FALSE;
                       END_IF;
                   END_REGION
               #S40_SET_EXCHANGE_BW_LOADER_LOAD:
                   REGION S40_SET_EXCHANGE_BW_LOADER_LOAD
                       IF #sInterface.SequenceReleased AND #sStepForward AND "AlwaysTRUE" THEN
                           #sCurrent_Step_NB := #S50_EXCHANGE_BW_LOADER_IN_PROGRESS;
                           #sCheck_Step_Condition := FALSE;
                       END_IF;
                   END_REGION
               #S50_EXCHANGE_BW_LOADER_IN_PROGRESS:
                   REGION S50_EXCHANGE_BW_LOADER_IN_PROGRESS
                       IF #sInterface.SequenceReleased AND #sStepForward AND (#iBwLoadDone OR "DB_BwLoaderExchange".Inputs.BwInErrorState <> 0) THEN
                           #sCurrent_Step_NB := #S60_EXCHANGE_BW_LOADER_ACQUIT;
                           #sCheck_Step_Condition := FALSE;
                       END_IF;
                   END_REGION
               #S60_EXCHANGE_BW_LOADER_ACQUIT:
                   REGION S60_EXCHANGE_BW_LOADER_ACQUIT
                       IF #sInterface.SequenceReleased AND #sStepForward AND "AlwaysTRUE" THEN
                           #sCurrent_Step_NB := #S195_JOB_DONE;
                           #sCheck_Step_Condition := FALSE;
                       END_IF;
                   END_REGION
               #S120_SHUTTLE_TO_BW_UNLOAD_POS_START_REQ:
                   REGION S120_SHUTTLE_TO_BW_UNLOAD_POS_START_REQ
                       IF #sInterface.SequenceReleased AND (#iShuttleMoving OR #iShuttleBwUnloadPos) THEN
                           #sCurrent_Step_NB := #S130_SHUTTLE_TO_BW_UNLOAD_POS_REACHED;
                           #sCheck_Step_Condition := FALSE;
                       END_IF;
                   END_REGION
               #S130_SHUTTLE_TO_BW_UNLOAD_POS_REACHED:
                   REGION S130_SHUTTLE_TO_BW_UNLOAD_POS_REACHED
                       IF #sInterface.SequenceReleased AND #sStepForward AND NOT #sShuttleStartReq AND #iShuttleBwUnloadPos AND "DB_BwLoaderExchange".Inputs.BwInErrorState = 0 THEN
                           #sCurrent_Step_NB := #S140_SET_EXCHANGE_BW_LOADER_UNLOAD;
                           #sCheck_Step_Condition := FALSE;
                       END_IF;
                   END_REGION
               #S140_SET_EXCHANGE_BW_LOADER_UNLOAD:
                   REGION S140_SET_EXCHANGE_BW_LOADER_UNLOAD
                       IF #sInterface.SequenceReleased AND #sStepForward AND "AlwaysTRUE" THEN
                           #sCurrent_Step_NB := #S150_EXCHANGE_BW_LOADER_IN_PROGRESS;
                           #sCheck_Step_Condition := FALSE;
                       END_IF;
                   END_REGION
               #S150_EXCHANGE_BW_LOADER_IN_PROGRESS:
                   REGION S150_EXCHANGE_BW_LOADER_IN_PROGRESS
                       IF #sInterface.SequenceReleased AND #sStepForward AND (#iBwUnloadDone OR "DB_BwLoaderExchange".Inputs.BwInErrorState <> 0) THEN
                           #sCurrent_Step_NB := #S160_EXCHANGE_BW_LOADER_ACQUIT;
                           #sCheck_Step_Condition := FALSE;
                       END_IF;
                   END_REGION
               #S160_EXCHANGE_BW_LOADER_ACQUIT:
                   REGION S160_EXCHANGE_BW_LOADER_ACQUIT
                       IF #sInterface.SequenceReleased AND #sStepForward AND "AlwaysTRUE" THEN
                           #sCurrent_Step_NB := #S195_JOB_DONE;
                           #sCheck_Step_Condition := FALSE;
                       END_IF;
                   END_REGION
               #S195_JOB_DONE:
                   REGION S95_JOB_DONE
                       IF NOT #iJobReq THEN
                           #sCurrent_Step_NB := #S00_INIT;
                           #sCheck_Step_Condition := FALSE;
                           #sInterface.JobDone := FALSE;
                       END_IF;
                   END_REGION
               ELSE
                   #sInterface.Error := TRUE;
           END_CASE;
       END_IF;
   END_REGION

   REGION Outputs Update
       #oShuttleStartReq := #sShuttleStartReq;
       #oShuttlePosSetPoint := #sShuttlePosSetPoint;
       #oBwLoadReq := #sBwLoadReq;
       #oBwUnloadReq := #sBwUnloadReq;
   END_REGION

   REGION Steps - Date and Time History
       IF #sHistory.Activation THEN
           IF #sHistory.Steps[0] <> #sCurrent_Step_NB THEN
               FOR #tIndex := 98 TO 0 BY -1 DO
                   #sHistory.Steps[#tIndex + 1] := #sHistory.Steps[#tIndex];
                   #sHistory.Date_Time[#tIndex + 1] := #sHistory.Date_Time[#tIndex];
               END_FOR;
               #sHistory.Steps[0] := #sCurrent_Step_NB;
               #sHistory.Date_Time[0] := #iPLC_DateAndTime;
           END_IF;
       END_IF;
   END_REGION

   REGION Steps Text
       #StepText(iErrorCode := #sCurrent_Step_NB,
                 oErrorText => #StepText.oErrorText);
   END_REGION
END_FUNCTION_BLOCK

FUNCTION_BLOCK "FB_BwControl"   // FB39, SCL
{ S7_Optimized_Access := 'TRUE' }
// stored: MemoryReserve 100, SetENOAutomatically false
   VAR_INPUT
      iStartSeqCond : Bool;   // Start Sequence Conditions
      iJobReq : Bool;   // Job Request - From Main
      iCtrlEnabled : Bool;   // Part Control Enable - Param or Condition
      iShuttleCtrlPos : Bool;   // Control Pos. Reached - Param
      iShuttleCtrlPosSetPoint : LReal;   // Control Pos. Setpoint - Param
      iExpectedCtrl : Bool;   // Expected result ctrl
      iBwPresence : Bool;   // Bw Presence - From DI
      iShuttleMoving : Bool;   // Shuttle is moving - From FB_LoaderAxis
      iShuttleInPos : Bool;   // Shuttle pos. reached - From FB_LoaderAxis
      iPLC_DateAndTime : DTL;
      iStepPause : Bool;
   END_VAR
   VAR_OUTPUT
      oShuttleStartReq { ExternalAccessible := 'False'; ExternalVisible := 'False'; ExternalWritable := 'False'} : Bool;   // Shuttle Start Order - To FB_LoaderAxis
      oShuttlePosSetPoint { ExternalAccessible := 'False'; ExternalVisible := 'False'; ExternalWritable := 'False'} : Real;   // Shuttle Position Setpoint - To FB_LoaderAxis
      oBwControlOK : Bool;   // Bw OK - To Main
      oBwControlNOK : Bool;   // Bw NOK - To Main
   END_VAR
   VAR
      sCurrent_Step_NB : Int;   // Active Step Number
      sCheck_Step_Condition : Bool;
      sOneStepForward : Bool;
      sRTOneStepForward : R_TRIG;
      sOneStepMode { S7_SetPoint := 'True'} : Bool;
      sStepForward : Bool;
      sInterface : "UDT_SequenceInterface";
      sShuttleStartReq { ExternalAccessible := 'False'; ExternalVisible := 'False'; ExternalWritable := 'False'} : Bool;
      sShuttlePosSetPoint { ExternalAccessible := 'False'; ExternalVisible := 'False'; ExternalWritable := 'False'} : Real;
      sMissingBwCtrl : Bool;
      sExtraBwCtrl : Bool;
      sPresenceBw : Bool;
      sBwControlOK : Bool;
      sBwControlNOK : Bool;
      sHistory : Struct
         Activation : Bool;
         Steps : Array[0..99] of Int;
         Date_Time : Array[0..99] of DTL;
      END_STRUCT;
      StepText : "FB_GetTextErrorCode";
   END_VAR
   VAR_TEMP
      tIndex : Int;   // Index
   END_VAR
   VAR CONSTANT
      S00_INIT : Int := 0;
      S10_CHECK_BW_PRESENCE_OPTION : Int := 10;
      S20_SHUTTLE_TO_BW_CTRL_POS_START_REQ : Int := 20;
      S30_SHUTTLE_TO_BW_CTRL_POS_REACHED : Int := 30;
      S40_WAIT_BW_CTRL_EXECUTION : Int := 40;
      S50_CHECK_BW_PRES_RESULT : Int := 50;
      S150_SET_BW_PRES_RESULT : Int := 150;
      S195_JOB_DONE : Int := 195;
   END_VAR
   // StepText.sCode_error[0].ErrorCode := 0;
   // StepText.sCode_error[1].ErrorCode := 10;
   // StepText.sCode_error[2].ErrorCode := 20;
   // StepText.sCode_error[3].ErrorCode := 30;
   // StepText.sCode_error[4].ErrorCode := 40;
   // StepText.sCode_error[5].ErrorCode := 50;
   // StepText.sCode_error[6].ErrorCode := 60;
   // StepText.sCode_error[7].ErrorCode := 70;
   // StepText.sCode_error[8].ErrorCode := 80;
   // StepText.sCode_error[9].ErrorCode := 90;
   // StepText.sCode_error[10].ErrorCode := 95;
BEGIN
   REGION Description header 
       //==================================================================================
       // POSALUX Swiss SA / (C) Copyright 2025
       //----------------------------------------------------------------------------------
       // Title: FB_BwControl
       // Comment/Function: 
       // Author: Fabien WALDT
       // Engineering: TIA Portal v17
       //----------------------------------------------------------------------------------
       // Change log table:
       // Version  | Date     | Expert in charge | Changes applied
       // ---------|----------|------------------|-----------------------------------------
       // 00.00.01 | 20250527 | WFA              | First released version
       // =================================================================================
   END_REGION

   REGION Define condition to start
       IF #iStartSeqCond THEN
           #sInterface.SequenceReleased := TRUE;
       ELSE
           // Standard sequencer controls
           #sInterface.SequenceReleased := FALSE;
           #sCurrent_Step_NB := #S00_INIT;
           #sInterface.SequenceRun := FALSE;
           #sInterface.JobDone := FALSE;
           #sCheck_Step_Condition := FALSE;

           // Dedicated sequencer controls
           #sShuttleStartReq := FALSE;
           #sShuttlePosSetPoint := 0.0;
           #sPresenceBw := FALSE;

           // Add specifics controls 
       END_IF;

       // Reset interface error
       IF #sInterface.Reset THEN
           #sInterface.Error := FALSE;
       END_IF;

       // Reset start when axis in position
       IF #iShuttleInPos THEN
           #sShuttleStartReq := FALSE;
       END_IF;

       // One step forward
       #sRTOneStepForward.CLK := #sOneStepForward;
       #sRTOneStepForward();
       #sStepForward := (NOT #sOneStepMode OR (#sOneStepMode AND #sRTOneStepForward.Q)) AND NOT #iStepPause;
       #sOneStepForward := FALSE;
   END_REGION

   REGION Sequence Function
       CASE #sCurrent_Step_NB OF
           #S00_INIT:
               REGION S00 INIT
                   #sCheck_Step_Condition := TRUE;
               END_REGION
           #S10_CHECK_BW_PRESENCE_OPTION:
               REGION S10_CHECK_BW_PRESENCE_OPTION
                   #sBwControlOK := FALSE;
                   #sBwControlNOK := FALSE;
                   #sMissingBwCtrl := FALSE;
                   #sExtraBwCtrl := FALSE;
                   #sCheck_Step_Condition := TRUE;
               END_REGION
           #S20_SHUTTLE_TO_BW_CTRL_POS_START_REQ:
               REGION S20_SHUTTLE_TO_BW_CTRL_POS_START_REQ
                   #sShuttleStartReq := NOT #iShuttleCtrlPos;
                   #sShuttlePosSetPoint := LREAL_TO_REAL(#iShuttleCtrlPosSetPoint);
                   #sCheck_Step_Condition := TRUE;
               END_REGION
           #S30_SHUTTLE_TO_BW_CTRL_POS_REACHED:
               REGION S30_SHUTTLE_TO_BW_CTRL_POS_REACHED
                   #sCheck_Step_Condition := TRUE;
               END_REGION
           #S40_WAIT_BW_CTRL_EXECUTION:
               REGION S40_WAIT_BW_CTRL_EXECUTION
                   #sPresenceBw := #iBwPresence;
                   #sCheck_Step_Condition := TRUE;
               END_REGION
           #S50_CHECK_BW_PRES_RESULT:
               REGION S50_CHECK_BW_PRES_RESULT
                   #sExtraBwCtrl := #sPresenceBw AND NOT #iExpectedCtrl;
                   #sMissingBwCtrl := NOT #sPresenceBw AND #iExpectedCtrl;
                   IF #sPresenceBw = #iExpectedCtrl THEN
                       #sBwControlOK := TRUE;
                       #sBwControlNOK := FALSE;
                   ELSE
                       #sBwControlOK := FALSE;
                       #sBwControlNOK := TRUE;
                   END_IF;
                   #sCheck_Step_Condition := TRUE;
               END_REGION
           #S150_SET_BW_PRES_RESULT:
               REGION S150_SET_BW_PRES_RESULT
                   #sBwControlOK := TRUE;
                   #sBwControlNOK := FALSE;
                   #sCheck_Step_Condition := TRUE;
               END_REGION
           #S195_JOB_DONE:
               REGION S195_JOB_DONE
                   #sInterface.JobDone := TRUE;
                   #sCheck_Step_Condition := TRUE;
               END_REGION
           ELSE:
               #sInterface.Error := TRUE;
       END_CASE;
   END_REGION

   REGION Sequence Next Step Condition
       IF #sCheck_Step_Condition THEN
           CASE #sCurrent_Step_NB OF
               #S00_INIT:
                   REGION S00 INIT
                       IF #sInterface.SequenceReleased AND #iJobReq THEN
                           #sCurrent_Step_NB := #S10_CHECK_BW_PRESENCE_OPTION;
                           #sInterface.SequenceRun := TRUE;
                           #sCheck_Step_Condition := FALSE;
                       ELSE
                           #sInterface.SequenceRun := FALSE;
                       END_IF;
                   END_REGION
               #S10_CHECK_BW_PRESENCE_OPTION:
                   REGION S10_CHECK_BW_PRESENCE_OPTION
                       IF #sInterface.SequenceReleased AND #sStepForward AND "DB_LoaderOptions".BwControl.UndrilledDrilledCtrlSeparate AND (NOT "DB_LoaderOptions".BwControl.Disabled OR NOT #iCtrlEnabled) THEN
                           #sCurrent_Step_NB := #S20_SHUTTLE_TO_BW_CTRL_POS_START_REQ;
                           #sCheck_Step_Condition := FALSE;
                       ELSIF #sInterface.SequenceReleased AND #sStepForward AND ("DB_LoaderOptions".BwControl.Disabled OR NOT #iCtrlEnabled) THEN
                           #sCurrent_Step_NB := #S150_SET_BW_PRES_RESULT;
                           #sCheck_Step_Condition := FALSE;
                       END_IF;
                   END_REGION
               #S20_SHUTTLE_TO_BW_CTRL_POS_START_REQ:
                   REGION S20_SHUTTLE_TO_BW_CTRL_POS_START_REQ
                       IF #sInterface.SequenceReleased AND (#iShuttleMoving OR #iShuttleCtrlPos) THEN
                           #sCurrent_Step_NB := #S30_SHUTTLE_TO_BW_CTRL_POS_REACHED;
                           #sCheck_Step_Condition := FALSE;
                       END_IF;
                   END_REGION
               #S30_SHUTTLE_TO_BW_CTRL_POS_REACHED:
                   REGION S30_SHUTTLE_TO_BW_CTRL_POS_REACHED
                       IF #sInterface.SequenceReleased AND #sStepForward AND NOT #sShuttleStartReq AND #iShuttleCtrlPos THEN
                           #sCurrent_Step_NB := #S40_WAIT_BW_CTRL_EXECUTION;
                           #sCheck_Step_Condition := FALSE;
                       END_IF;
                   END_REGION
               #S40_WAIT_BW_CTRL_EXECUTION:
                   REGION S40_WAIT_BW_CTRL_EXECUTION
                       IF #sInterface.SequenceReleased AND #sStepForward AND "AlwaysTRUE" THEN
                           #sCurrent_Step_NB := #S50_CHECK_BW_PRES_RESULT;
                           #sCheck_Step_Condition := FALSE;
                       END_IF;
                   END_REGION
               #S50_CHECK_BW_PRES_RESULT:
                   REGION S50_CHECK_BW_PRES_RESULT
                       IF #sInterface.SequenceReleased AND #sStepForward AND "AlwaysTRUE" THEN
                           #sCurrent_Step_NB := #S195_JOB_DONE;
                           #sCheck_Step_Condition := FALSE;
                       END_IF;
                   END_REGION
               #S150_SET_BW_PRES_RESULT:
                   REGION S150_SET_BW_PRES_RESULT
                       IF #sInterface.SequenceReleased AND #sStepForward AND "AlwaysTRUE" THEN
                           #sCurrent_Step_NB := #S195_JOB_DONE;
                           #sCheck_Step_Condition := FALSE;
                       END_IF;
                   END_REGION
               #S195_JOB_DONE:
                   REGION S195_JOB_DONE
                       IF NOT #iJobReq THEN
                           #sCurrent_Step_NB := #S00_INIT;
                           #sCheck_Step_Condition := FALSE;
                           #sInterface.JobDone := FALSE;
                       END_IF;
                   END_REGION
               ELSE
                   #sInterface.Error := TRUE;
           END_CASE;
       END_IF;
   END_REGION

   REGION Outputs Update
       #oShuttleStartReq := #sShuttleStartReq;
       #oShuttlePosSetPoint := #sShuttlePosSetPoint;
       #oBwControlOK := #sBwControlOK;
       #oBwControlNOK := #sBwControlNOK;
   END_REGION

   REGION Steps - Date and Time History
       IF #sHistory.Activation THEN
           IF #sHistory.Steps[0] <> #sCurrent_Step_NB THEN
               FOR #tIndex := 98 TO 0 BY -1 DO
                   #sHistory.Steps[#tIndex + 1] := #sHistory.Steps[#tIndex];
                   #sHistory.Date_Time[#tIndex + 1] := #sHistory.Date_Time[#tIndex];
               END_FOR;
               #sHistory.Steps[0] := #sCurrent_Step_NB;
               #sHistory.Date_Time[0] := #iPLC_DateAndTime;
           END_IF;
       END_IF;
   END_REGION

   REGION Steps Text
       #StepText(iErrorCode := #sCurrent_Step_NB,
                 oErrorText => #StepText.oErrorText);
   END_REGION
END_FUNCTION_BLOCK

FUNCTION_BLOCK "FB_Consecutive"   // FB90, SCL
{ S7_Optimized_Access := 'TRUE' }
// stored: MemoryReserve 100, SetENOAutomatically false
   VAR_INPUT
      iReset : Bool;
      iGoodEntry : Bool;
      iBadEntry : Bool;
      iPresetValue : Int;
   END_VAR
   VAR_OUTPUT
      oConsecutiveError : Bool;
   END_VAR
   VAR
      sConsecutiveCounter : Int;
      sRT_GoodEntry : R_TRIG;
      sRT_BadEntry { S7_SetPoint := 'True'} : R_TRIG;
   END_VAR
BEGIN
   REGION Description header 
       //==================================================================================
       // POSALUX Swiss SA / (C) Copyright 2026
       //----------------------------------------------------------------------------------
       // Title: FB_Consecutive
       // Comment/Function: 
       // Author: Fabien WALDT
       // Engineering: TIA Portal v20
       //----------------------------------------------------------------------------------
       // Change log table:
       // Version  | Date     | Expert in charge | Changes applied
       // ---------|----------|------------------|-----------------------------------------
       // 00.00.01 | 20260401 | WFA              | First released version
       // =================================================================================
   END_REGION

   REGION R_Trig
       #sRT_GoodEntry(CLK := #iGoodEntry);
       #sRT_BadEntry(CLK := #iBadEntry);
   END_REGION

   REGION Consecutive Counter
       IF #sRT_GoodEntry.Q OR #iReset THEN
           #oConsecutiveError := FALSE;
           #sConsecutiveCounter := 0;
       END_IF;

       IF #sRT_BadEntry.Q THEN
           #sConsecutiveCounter := #sConsecutiveCounter + 1;
       END_IF;

       IF #sConsecutiveCounter >= #iPresetValue THEN
           #oConsecutiveError := TRUE;
       END_IF;
   END_REGION
END_FUNCTION_BLOCK

FUNCTION_BLOCK "FB_Blowing"   // FB63, SCL
{ S7_Optimized_Access := 'TRUE' }
// stored: AutoNumber false, MemoryReserve 100, SetENOAutomatically false
   VAR_INPUT
      iStartSeqCond : Bool;   // Start Sequence Conditions
      iJobReq : Bool;   // Job Request - From Main
      iShuttleBlowingPos : Bool;   // Load/Unload Pos. Reached - Param
      iShuttleBlowingPosSetPoint : LReal;   // Load/Unload Pos. Setpoint - Param
      iAxisV_BlowingPos : Bool;
      iAxisV_BlowingPosSetPoint : LReal;
      iAxisW_SafePos : Bool;
      iAxisW_SafePosSetPoint : LReal;
      iAxisW_BlowingPos : Bool;
      iAxisW_BlowingPosSetPoint : LReal;
      iShuttleMoving : Bool;   // Shuttle is moving - From FB_LoaderAxis
      iShuttleInPos : Bool;   // Shuttle pos. reached - From FB_LoaderAxis
      iAxisV_Moving : Bool;   // Shuttle is moving
      iAxisV_InPos : Bool;
      iAxisW_Moving { ExternalAccessible := 'False'; ExternalVisible := 'False'; ExternalWritable := 'False'} : Bool;   // Shuttle is moving
      iAxisW_InPos : Bool;
      iBlowingTime : Time;
      iPLC_DateAndTime : DTL;
      iStepPause : Bool;
   END_VAR
   VAR_OUTPUT
      oShuttleStartReq { ExternalAccessible := 'False'; ExternalVisible := 'False'; ExternalWritable := 'False'} : Bool;   // Shuttle Start Order - To FB_LoaderAxis
      oShuttlePosSetPoint { ExternalAccessible := 'False'; ExternalVisible := 'False'; ExternalWritable := 'False'} : Real;   // Shuttle Position Setpoint - To FB_LoaderAxis
      oAxisV_StartReq : Bool;
      oAxisV_PosSetPoint : Real;
      oAxisW_StartReq : Bool;
      oAxisW_PosSetPoint : Real;
      oBlowingReq : Bool;
   END_VAR
   VAR
      sCurrent_Step_NB : Int;   // Active Step Number
      sCheck_Step_Condition : Bool;
      sOneStepForward : Bool;
      sRTOneStepForward : R_TRIG;
      sOneStepMode { S7_SetPoint := 'True'} : Bool;
      sStepForward : Bool;
      sInterface : "UDT_SequenceInterface";
      sShuttleStartReq { ExternalAccessible := 'False'; ExternalVisible := 'False'; ExternalWritable := 'False'} : Bool;
      sShuttlePosSetPoint { ExternalAccessible := 'False'; ExternalVisible := 'False'; ExternalWritable := 'False'} : Real;
      sAxisV_StartReq : Bool;
      sAxisV_PosSetPoint : Real;
      sAxisW_StartReq : Bool;
      sAxisW_PosSetPoint : Real;
      sBlowingReq : Bool;   // Drilled Part To Unload - From FB_Position
      sBlowingTimerStart : Bool;
      sBlowingTimer : TP_TIME;
      sFT_BlowingTimer { S7_SetPoint := 'True'} : F_TRIG;
      sHistory : Struct
         Activation : Bool;
         Steps : Array[0..99] of Int;
         Date_Time : Array[0..99] of DTL;
      END_STRUCT;
      StepText : "FB_GetTextErrorCode";
   END_VAR
   VAR_TEMP
      tIndex : Int;   // Index
   END_VAR
   VAR CONSTANT
      S00_INIT : Int := 0;
      S10_CHECK_BLOWING_OPTION : Int := 10;
      S20_SHUTTLE_TO_BLOWING_POS_START_REQ : Int := 20;
      S30_SHUTTLE_TO_BLOWING_POS_REACHED : Int := 30;
      S40_AXIS_W_TO_SAFE_POS_START_REQ : Int := 40;
      S50_AXIS_W_TO_SAFE_POS_REACHED : Int := 50;
      S60_AXIS_V_TO_BLOWING_POS_START_REQ : Int := 60;
      S70_AXIS_V_TO_BLOWING_POS_REACHED : Int := 70;
      S80_AXIS_W_TO_BLOWING_POS_START_REQ : Int := 80;
      S90_AXIS_W_TO_BLOWING_POS_REACHED : Int := 90;
      S100_BLOWING_TIMER_START_REQ : Int := 100;
      S195_JOB_DONE : Int := 195;
   END_VAR
   // StepText.sCode_error[0].ErrorCode := 0;
   // StepText.sCode_error[1].ErrorCode := 10;
   // StepText.sCode_error[2].ErrorCode := 20;
   // StepText.sCode_error[3].ErrorCode := 30;
   // StepText.sCode_error[4].ErrorCode := 40;
   // StepText.sCode_error[5].ErrorCode := 50;
   // StepText.sCode_error[6].ErrorCode := 60;
   // StepText.sCode_error[7].ErrorCode := 70;
   // StepText.sCode_error[8].ErrorCode := 80;
   // StepText.sCode_error[9].ErrorCode := 90;
   // StepText.sCode_error[10].ErrorCode := 95;
BEGIN
   REGION Description header 
       //==================================================================================
       // POSALUX Swiss SA / (C) Copyright 2025
       //----------------------------------------------------------------------------------
       // Title: FB_Blowing
       // Comment/Function: 
       // Author: Fabien WALDT
       // Engineering: TIA Portal v17
       //----------------------------------------------------------------------------------
       // Change log table:
       // Version  | Date     | Expert in charge | Changes applied
       // ---------|----------|------------------|-----------------------------------------
       // 00.00.01 | 20250527 | WFA              | First released version
       // =================================================================================
   END_REGION

   REGION Define condition to start
       IF #iStartSeqCond THEN
           #sInterface.SequenceReleased := TRUE;
       ELSE
           // Standard sequencer controls
           #sInterface.SequenceReleased := FALSE;
           #sCurrent_Step_NB := #S00_INIT;
           #sInterface.SequenceRun := FALSE;
           #sInterface.JobDone := FALSE;
           #sCheck_Step_Condition := FALSE;

           // Dedicated sequencer controls
           #sShuttleStartReq := FALSE;
           #sShuttlePosSetPoint := 0.0;
           #sAxisV_StartReq := FALSE;
           #sAxisV_PosSetPoint := 0.0;
           #sAxisW_StartReq := FALSE;
           #sAxisW_PosSetPoint := 0.0;
           #sBlowingReq := FALSE;
           #sBlowingTimerStart := FALSE;

           // Add specifics controls 
       END_IF;

       // Reset interface error
       IF #sInterface.Reset THEN
           #sInterface.Error := FALSE;
       END_IF;

       // Reset start when axis in position
       IF #iShuttleInPos THEN
           #sShuttleStartReq := FALSE;
       END_IF;
       IF #iAxisV_InPos THEN
           #sAxisV_StartReq := FALSE;
       END_IF;
       IF #iAxisW_InPos THEN
           #sAxisW_StartReq := FALSE;
       END_IF;

       // One step forward
       #sRTOneStepForward.CLK := #sOneStepForward;
       #sRTOneStepForward();
       #sStepForward := (NOT #sOneStepMode OR (#sOneStepMode AND #sRTOneStepForward.Q)) AND NOT #iStepPause;
       #sOneStepForward := FALSE;

       // Action only true in dedicated steps
       #sBlowingReq := FALSE;

       // Blowing Timer
       #sBlowingTimer(IN := #sBlowingTimerStart AND #sStepForward,
                      PT := #iBlowingTime);

       #sFT_BlowingTimer(CLK := #sBlowingTimer.Q);

       #sBlowingReq := #sBlowingTimer.Q;
   END_REGION

   REGION Sequence Function
       CASE #sCurrent_Step_NB OF
           #S00_INIT:
               REGION S00 INIT
                   #sCheck_Step_Condition := TRUE;
               END_REGION
           #S10_CHECK_BLOWING_OPTION:
               REGION S10_CHECK_BLOWING_OPTION
                   #sCheck_Step_Condition := TRUE;
               END_REGION
           #S20_SHUTTLE_TO_BLOWING_POS_START_REQ:
               REGION S20_SHUTTLE_TO_BLOWING_POS_START_REQ
                   #sShuttleStartReq := NOT #iShuttleBlowingPos;
                   #sShuttlePosSetPoint := LREAL_TO_REAL(#iShuttleBlowingPosSetPoint);
                   #sCheck_Step_Condition := TRUE;
               END_REGION
           #S30_SHUTTLE_TO_BLOWING_POS_REACHED:
               REGION S30_SHUTTLE_TO_BLOWING_POS_REACHED
                   #sCheck_Step_Condition := TRUE;
               END_REGION
           #S40_AXIS_W_TO_SAFE_POS_START_REQ:
               REGION S40_AXIS_W_TO_SAFE_POS_START_REQ
                   #sAxisW_StartReq := NOT #iAxisW_SafePos;
                   #sAxisW_PosSetPoint := LREAL_TO_REAL(#iAxisW_SafePosSetPoint);
                   #sCheck_Step_Condition := TRUE;
               END_REGION
           #S50_AXIS_W_TO_SAFE_POS_REACHED:
               REGION S50_AXIS_W_TO_SAFE_POS_REACHED
                   #sCheck_Step_Condition := TRUE;
               END_REGION
           #S60_AXIS_V_TO_BLOWING_POS_START_REQ:
               REGION S60_AXIS_V_TO_BLOWING_POS_START_REQ
                   #sAxisV_StartReq := NOT #iAxisV_BlowingPos;
                   #sAxisV_PosSetPoint := LREAL_TO_REAL(#iAxisV_BlowingPosSetPoint);
                   #sCheck_Step_Condition := TRUE;
               END_REGION
           #S70_AXIS_V_TO_BLOWING_POS_REACHED:
               REGION S70_AXIS_V_TO_BLOWING_POS_REACHED
                   #sCheck_Step_Condition := TRUE;
               END_REGION
           #S80_AXIS_W_TO_BLOWING_POS_START_REQ:
               REGION S80_AXIS_W_TO_BLOWING_POS_START_REQ
                   #sAxisW_StartReq := NOT #iAxisW_BlowingPos;
                   #sAxisW_PosSetPoint := LREAL_TO_REAL(#iAxisW_BlowingPosSetPoint);
                   #sCheck_Step_Condition := TRUE;
               END_REGION
           #S90_AXIS_W_TO_BLOWING_POS_REACHED:
               REGION S90_AXIS_W_TO_BLOWING_POS_REACHED
                   #sCheck_Step_Condition := TRUE;
               END_REGION
           #S100_BLOWING_TIMER_START_REQ:
               REGION S100_BLOWING TIMER_START_REQ
                   #sBlowingTimerStart := TRUE;
                   #sCheck_Step_Condition := TRUE;
               END_REGION
           #S195_JOB_DONE:
               REGION S195_JOB_DONE
                   #sBlowingTimerStart := FALSE;
                   #sInterface.JobDone := TRUE;
                   #sCheck_Step_Condition := TRUE;
               END_REGION
           ELSE:
               #sInterface.Error := TRUE;
       END_CASE;
   END_REGION

   REGION Sequence Next Step Condition
       IF #sCheck_Step_Condition THEN
           CASE #sCurrent_Step_NB OF
               #S00_INIT:
                   REGION S00 INIT
                       IF #sInterface.SequenceReleased AND #iJobReq THEN
                           #sCurrent_Step_NB := #S10_CHECK_BLOWING_OPTION;
                           #sInterface.SequenceRun := TRUE;
                           #sCheck_Step_Condition := FALSE;
                       ELSE
                           #sInterface.SequenceRun := FALSE;
                       END_IF;
                   END_REGION
               #S10_CHECK_BLOWING_OPTION:
                   REGION S10_CHECK_BLOWING_OPTION
                       IF #sInterface.SequenceReleased AND #sStepForward AND "DB_LoaderOptions".Blowing.Inside AND NOT "DB_LoaderOptions".Blowing.Disabled  THEN
                           #sCurrent_Step_NB := #S20_SHUTTLE_TO_BLOWING_POS_START_REQ;
                           #sCheck_Step_Condition := FALSE;
                       ELSIF #sInterface.SequenceReleased AND #sStepForward AND (NOT "DB_LoaderOptions".Blowing.Inside OR NOT "DB_LoaderOptions".Blowing.Disabled)  THEN
                           #sCurrent_Step_NB := #S195_JOB_DONE;
                           #sCheck_Step_Condition := FALSE;
                       END_IF;
                   END_REGION
               #S20_SHUTTLE_TO_BLOWING_POS_START_REQ:
                   REGION S20_SHUTTLE_TO_BLOWING_POS_START_REQ
                       IF #sInterface.SequenceReleased AND (#iShuttleMoving OR #iShuttleBlowingPos) THEN
                           #sCurrent_Step_NB := #S30_SHUTTLE_TO_BLOWING_POS_REACHED;
                           #sCheck_Step_Condition := FALSE;
                       END_IF;
                   END_REGION
               #S30_SHUTTLE_TO_BLOWING_POS_REACHED:
                   REGION S30_SHUTTLE_TO_BLOWING_POS_REACHED
                       IF #sInterface.SequenceReleased AND #sStepForward AND NOT #sShuttleStartReq AND #iShuttleBlowingPos THEN
                           #sCurrent_Step_NB := #S40_AXIS_W_TO_SAFE_POS_START_REQ;
                           #sCheck_Step_Condition := FALSE;
                       END_IF;
                   END_REGION
               #S40_AXIS_W_TO_SAFE_POS_START_REQ:
                   REGION S40_AXIS_W_TO_SAFE_POS_START_REQ
                       IF #sInterface.SequenceReleased AND (#iAxisW_Moving OR #iAxisW_SafePos) THEN
                           #sCurrent_Step_NB := #S50_AXIS_W_TO_SAFE_POS_REACHED;
                           #sCheck_Step_Condition := FALSE;
                       END_IF;
                   END_REGION
               #S50_AXIS_W_TO_SAFE_POS_REACHED:
                   REGION S50_AXIS_W_TO_SAFE_POS_REACHED
                       IF #sInterface.SequenceReleased AND #sStepForward AND NOT #sAxisW_StartReq AND #iAxisW_SafePos THEN
                           #sCurrent_Step_NB := #S60_AXIS_V_TO_BLOWING_POS_START_REQ;
                           #sCheck_Step_Condition := FALSE;
                       END_IF;
                   END_REGION
               #S60_AXIS_V_TO_BLOWING_POS_START_REQ:
                   REGION S60_AXIS_V_TO_BLOWING_POS_START_REQ
                       IF #sInterface.SequenceReleased AND #sStepForward AND (#iAxisV_Moving OR #iAxisV_BlowingPos) THEN
                           #sCurrent_Step_NB := #S70_AXIS_V_TO_BLOWING_POS_REACHED;
                           #sCheck_Step_Condition := FALSE;
                       END_IF;
                   END_REGION
               #S70_AXIS_V_TO_BLOWING_POS_REACHED:
                   REGION S70_AXIS_V_TO_BLOWING_POS_REACHED
                       IF #sInterface.SequenceReleased AND #sStepForward AND NOT #sAxisV_StartReq AND #iAxisV_BlowingPos THEN
                           #sCurrent_Step_NB := #S80_AXIS_W_TO_BLOWING_POS_START_REQ;
                           #sCheck_Step_Condition := FALSE;
                       END_IF;
                   END_REGION
               #S80_AXIS_W_TO_BLOWING_POS_START_REQ:
                   REGION S80_AXIS_W_TO_BLOWING_POS_START_REQ
                       IF #sInterface.SequenceReleased AND (#iAxisW_Moving OR #iAxisW_BlowingPos) THEN
                           #sCurrent_Step_NB := #S90_AXIS_W_TO_BLOWING_POS_REACHED;
                           #sCheck_Step_Condition := FALSE;
                       END_IF;
                   END_REGION
               #S90_AXIS_W_TO_BLOWING_POS_REACHED:
                   REGION S90_AXIS_W_TO_BLOWING_POS_REACHED
                       IF #sInterface.SequenceReleased AND #sStepForward AND NOT #sAxisW_StartReq AND #iAxisW_BlowingPos THEN
                           #sCurrent_Step_NB := #S100_BLOWING_TIMER_START_REQ;
                           #sCheck_Step_Condition := FALSE;
                       END_IF;
                   END_REGION
               #S100_BLOWING_TIMER_START_REQ:
                   REGION S100_BLOWING_TIMER_START_REQ
                       IF #sInterface.SequenceReleased AND #sStepForward AND #sFT_BlowingTimer.Q THEN
                           #sCurrent_Step_NB := #S195_JOB_DONE;
                           #sCheck_Step_Condition := FALSE;
                       END_IF;
                   END_REGION
               #S195_JOB_DONE:
                   REGION S95_JOB_DONE
                       IF NOT #iJobReq THEN
                           #sCurrent_Step_NB := #S00_INIT;
                           #sCheck_Step_Condition := FALSE;
                           #sInterface.JobDone := FALSE;
                       END_IF;
                   END_REGION
               ELSE
                   #sInterface.Error := TRUE;
           END_CASE;
       END_IF;
   END_REGION

   REGION Outputs Update
       #oShuttleStartReq := #sShuttleStartReq;
       #oShuttlePosSetPoint := #sShuttlePosSetPoint;
       #oAxisV_StartReq := #sAxisV_StartReq;
       #oAxisV_PosSetPoint := #sAxisV_PosSetPoint;
       #oAxisW_StartReq := #sAxisW_StartReq;
       #oAxisW_PosSetPoint := #sAxisW_PosSetPoint;
       #oBlowingReq := #sBlowingReq;
   END_REGION

   REGION Steps - Date and Time History
       IF #sHistory.Activation THEN
           IF #sHistory.Steps[0] <> #sCurrent_Step_NB THEN
               FOR #tIndex := 98 TO 0 BY -1 DO
                   #sHistory.Steps[#tIndex + 1] := #sHistory.Steps[#tIndex];
                   #sHistory.Date_Time[#tIndex + 1] := #sHistory.Date_Time[#tIndex];
               END_FOR;
               #sHistory.Steps[0] := #sCurrent_Step_NB;
               #sHistory.Date_Time[0] := #iPLC_DateAndTime;
           END_IF;
       END_IF;
   END_REGION

   REGION Steps Text
       #StepText(iErrorCode := #sCurrent_Step_NB,
                 oErrorText => #StepText.oErrorText);
   END_REGION
END_FUNCTION_BLOCK

FUNCTION_BLOCK "FB_ActControl"   // FB45, SCL
{ S7_Optimized_Access := 'TRUE' }
// stored: MemoryReserve 100, SetENOAutomatically false
   VAR_INPUT
      iStartSeqCond : Bool;   // Start Sequence Conditions
      iJobReq : Bool;   // Job Request - From Main
      iShuttleModeAutoPos : Bool;   // Load/Unload Manu Pos. Reached - Param
      iShuttleModeAutoPosSetPoint : LReal;   // Load/Unload Manu Pos. Setpoint - Param
      iShuttleModeSemiAutoPos : Bool;   // Load/Unload Manu Pos. Reached - Param
      iShuttleModeSemiAutoPosSetPoint : LReal;   // Load/Unload Manu Pos. Setpoint - Param
      iShuttleMoving : Bool;   // Shuttle is moving - From FB_LoaderAxis
      iShuttleInPos : Bool;   // Shuttle pos. reached - From FB_LoaderAxis
      iModeAutoPosCondition : Bool;
      iModeSemiAutoPosCondition : Bool;
      iNoStopCondition : Bool;
      iOperatorCycleRestart : Bool;
      iNC_Stopped : Bool;
      iNC_Running : Bool;
      iMissingPart : Bool;
      iExtraPart : Bool;
      iPLC_DateAndTime : DTL;
      iStepPause : Bool;
   END_VAR
   VAR_OUTPUT
      oShuttleStartReq { ExternalAccessible := 'False'; ExternalVisible := 'False'; ExternalWritable := 'False'} : Bool;   // Shuttle Start Order - To FB_LoaderAxis
      oShuttlePosSetPoint { ExternalAccessible := 'False'; ExternalVisible := 'False'; ExternalWritable := 'False'} : Real;   // Shuttle Position Setpoint - To FB_LoaderAxis
      oStopNC_Req : Bool;
      oRestartNC_Req : Bool;
      oRestartStep : Bool;
      oContinuationStep : Bool;
      oMsgMissingPart : Bool;
      oMsgExtraPart : Bool;
   END_VAR
   VAR
      sCurrent_Step_NB : Int;   // Active Step Number
      sCheck_Step_Condition : Bool;
      sOneStepForward : Bool;
      sRTOneStepForward : R_TRIG;
      sOneStepMode { S7_SetPoint := 'True'} : Bool;
      sStepForward : Bool;
      sInterface : "UDT_SequenceInterface";
      sShuttleStartReq { ExternalAccessible := 'False'; ExternalVisible := 'False'; ExternalWritable := 'False'} : Bool;
      sShuttlePosSetPoint { ExternalAccessible := 'False'; ExternalVisible := 'False'; ExternalWritable := 'False'} : Real;
      sStopNC_Req : Bool;
      sRestartNC_Req : Bool;
      sRestartStep : Bool;
      sContinuationStep : Bool;
      sMsgMissingPart : Bool;
      sMsgExtraPart : Bool;
      sHistory : Struct
         Activation : Bool;
         Steps : Array[0..99] of Int;
         Date_Time : Array[0..99] of DTL;
      END_STRUCT;
      StepText : "FB_GetTextErrorCode";
   END_VAR
   VAR_TEMP
      tIndex : Int;   // Index
   END_VAR
   VAR CONSTANT
      S00_INIT : Int := 0;
      S10_CHECK_ACT_CTRL_OPTION : Int := 10;
      S20_SHUTTLE_TO_STOP_CYCLE_POS_START_REQ : Int := 20;
      S30_SHUTTLE_TO_STOP_CYCLE_POS_REACHED : Int := 30;
      S40_STOP_CYCLE : Int := 40;
      S50_WAIT_OPERATOR_RESTART : Int := 50;
      S60_NC_RESTART : Int := 60;
      S70_UPDATE_NEXT_STEP : Int := 70;
      S120_SHUTTLE_TO_EXT_LOAD_UNLOAD_POS_START_REQ : Int := 120;
      S130_SHUTTLE_TO_EXT_LOAD_UNLOAD_POS_REACHED : Int := 130;
      S140_STOP_CYCLE : Int := 140;
      S150_WAIT_OPERATOR_RESTART : Int := 150;
      S160_NC_RESTART : Int := 160;
      S170_UPDATE_NEXT_STEP : Int := 170;
      S270_UPDATE_NEXT_STEP : Int := 270;
      S295_JOB_DONE : Int := 295;
   END_VAR
   // StepText.sCode_error[0].ErrorCode := 0;
   // StepText.sCode_error[1].ErrorCode := 10;
   // StepText.sCode_error[2].ErrorCode := 20;
   // StepText.sCode_error[3].ErrorCode := 30;
   // StepText.sCode_error[4].ErrorCode := 40;
   // StepText.sCode_error[5].ErrorCode := 50;
   // StepText.sCode_error[6].ErrorCode := 60;
   // StepText.sCode_error[7].ErrorCode := 70;
   // StepText.sCode_error[8].ErrorCode := 80;
   // StepText.sCode_error[9].ErrorCode := 90;
   // StepText.sCode_error[10].ErrorCode := 95;
BEGIN
   REGION Description header 
       //==================================================================================
       // POSALUX Swiss SA / (C) Copyright 2025
       //----------------------------------------------------------------------------------
       // Title: FB_ActControl
       // Comment/Function: 
       // Author: Fabien WALDT
       // Engineering: TIA Portal v17
       //----------------------------------------------------------------------------------
       // Change log table:
       // Version  | Date     | Expert in charge | Changes applied
       // ---------|----------|------------------|-----------------------------------------
       // 00.00.01 | 20250527 | WFA              | First released version
       // =================================================================================
   END_REGION

   REGION Define condition to start
       IF #iStartSeqCond THEN
           #sInterface.SequenceReleased := TRUE;
       ELSE
           // Standard sequencer controls
           #sInterface.SequenceReleased := FALSE;
           #sCurrent_Step_NB := #S00_INIT;
           #sInterface.SequenceRun := FALSE;
           #sInterface.JobDone := FALSE;
           #sCheck_Step_Condition := FALSE;

           // Dedicated sequencer controls
           #sShuttleStartReq := FALSE;
           #sShuttlePosSetPoint := 0.0;
           #sStopNC_Req := FALSE;
           #sRestartNC_Req := FALSE;
           #sRestartStep := FALSE;
           #sContinuationStep := FALSE;


           // Add specifics controls 
       END_IF;

       // Reset interface error
       IF #sInterface.Reset THEN
           #sInterface.Error := FALSE;
       END_IF;

       // Reset start when axis in position
       IF #iShuttleInPos THEN
           #sShuttleStartReq := FALSE;
       END_IF;

       // One step forward
       #sRTOneStepForward.CLK := #sOneStepForward;
       #sRTOneStepForward();
       #sStepForward := (NOT #sOneStepMode OR (#sOneStepMode AND #sRTOneStepForward.Q)) AND NOT #iStepPause;
       #sOneStepForward := FALSE;

       // Action only true in dedicated steps
       #sStopNC_Req := FALSE;
       #sRestartNC_Req := FALSE;
   END_REGION

   REGION Sequence Function
       CASE #sCurrent_Step_NB OF
           #S00_INIT:
               REGION S00 INIT
                   #sCheck_Step_Condition := TRUE;
                   #sMsgMissingPart := FALSE;
                   #sMsgExtraPart := FALSE;
               END_REGION
           #S10_CHECK_ACT_CTRL_OPTION:
               REGION S10_CHECK_ACT_CTRL_OPTION
                   #sCheck_Step_Condition := TRUE;
               END_REGION
           #S20_SHUTTLE_TO_STOP_CYCLE_POS_START_REQ:
               REGION S20_SHUTTLE_TO_STOP_CYCLE_POS_START_REQ
                   #sShuttleStartReq := NOT #iShuttleModeAutoPos;
                   #sShuttlePosSetPoint := LREAL_TO_REAL(#iShuttleModeAutoPosSetPoint);
                   #sCheck_Step_Condition := TRUE;
               END_REGION
           #S30_SHUTTLE_TO_STOP_CYCLE_POS_REACHED:
               REGION S30_SHUTTLE_TO_STOP_CYCLE_POS_REACHED
                   #sCheck_Step_Condition := TRUE;
               END_REGION
           #S40_STOP_CYCLE:
               REGION S40_STOP_CYCLE
                   #sStopNC_Req := TRUE;
                   #sMsgMissingPart := #iMissingPart;
                   #sMsgExtraPart := #iExtraPart;
                   #sCheck_Step_Condition := TRUE;
               END_REGION
           #S50_WAIT_OPERATOR_RESTART:
               REGION S50_WAIT_OPERATOR_RESTART
                   #sCheck_Step_Condition := TRUE;
               END_REGION
           #S60_NC_RESTART:
               REGION S60_NC_RESTART
                   #sRestartNC_Req := TRUE;
                   #sCheck_Step_Condition := TRUE;
               END_REGION
           #S70_UPDATE_NEXT_STEP:
               REGION S70_UPDATE_NEXT_STEP
                   #sRestartStep := TRUE;
                   #sContinuationStep := FALSE;
                   #sCheck_Step_Condition := TRUE;
               END_REGION

           #S120_SHUTTLE_TO_EXT_LOAD_UNLOAD_POS_START_REQ:
               REGION S120_SHUTTLE_TO_EXT_LOAD_UNLOAD_POS_START_REQ
                   #sShuttleStartReq := NOT #iShuttleModeSemiAutoPos;
                   #sShuttlePosSetPoint := LREAL_TO_REAL(#iShuttleModeSemiAutoPosSetPoint);
                   #sCheck_Step_Condition := TRUE;
               END_REGION
           #S130_SHUTTLE_TO_EXT_LOAD_UNLOAD_POS_REACHED:
               REGION S130_SHUTTLE_TO_EXT_LOAD_UNLOAD_POS_REACHED
                   #sCheck_Step_Condition := TRUE;
               END_REGION
           #S140_STOP_CYCLE:
               REGION S140_STOP_CYCLE
                   #sStopNC_Req := TRUE;
                   #sMsgMissingPart := #iMissingPart;
                   #sMsgExtraPart := #iExtraPart;
                   #sCheck_Step_Condition := TRUE;
               END_REGION
           #S150_WAIT_OPERATOR_RESTART:
               REGION S150_WAIT_OPERATOR_RESTART
                   #sCheck_Step_Condition := TRUE;
               END_REGION
           #S160_NC_RESTART:
               REGION S160_NC_RESTART
                   #sRestartNC_Req := TRUE;
                   #sCheck_Step_Condition := TRUE;
               END_REGION
           #S170_UPDATE_NEXT_STEP:
               REGION S170_UPDATE_NEXT_STEP
                   #sRestartStep := TRUE;
                   #sContinuationStep := FALSE;
                   #sCheck_Step_Condition := TRUE;
               END_REGION

           #S270_UPDATE_NEXT_STEP:
               REGION S270_UPDATE_NEXT_STEP
                   #sRestartStep := FALSE;
                   #sContinuationStep := TRUE;
                   #sCheck_Step_Condition := TRUE;
               END_REGION

           #S295_JOB_DONE:
               REGION S295_JOB_DONE
                   #sInterface.JobDone := TRUE;
                   #sCheck_Step_Condition := TRUE;
               END_REGION
           ELSE:
               #sInterface.Error := TRUE;
       END_CASE;
   END_REGION

   REGION Sequence Next Step Condition
       IF #sCheck_Step_Condition THEN
           CASE #sCurrent_Step_NB OF
               #S00_INIT:
                   REGION S00 INIT
                       IF #sInterface.SequenceReleased AND #iJobReq THEN
                           #sCurrent_Step_NB := #S10_CHECK_ACT_CTRL_OPTION;
                           #sInterface.SequenceRun := TRUE;
                           #sCheck_Step_Condition := FALSE;
                       ELSE
                           #sInterface.SequenceRun := FALSE;
                       END_IF;
                   END_REGION
               #S10_CHECK_ACT_CTRL_OPTION:
                   REGION S10_CHECK_ACT_CTRL_OPTION
                       IF #sInterface.SequenceReleased AND #sStepForward AND #iModeAutoPosCondition AND NOT #iModeSemiAutoPosCondition AND NOT #iNoStopCondition THEN
                           #sCurrent_Step_NB := #S20_SHUTTLE_TO_STOP_CYCLE_POS_START_REQ;
                           #sCheck_Step_Condition := FALSE;
                       ELSIF #sInterface.SequenceReleased AND #sStepForward AND NOT #iModeAutoPosCondition AND #iModeSemiAutoPosCondition AND NOT #iNoStopCondition THEN
                           #sCurrent_Step_NB := #S120_SHUTTLE_TO_EXT_LOAD_UNLOAD_POS_START_REQ;
                           #sCheck_Step_Condition := FALSE;
                       ELSIF #sInterface.SequenceReleased AND #sStepForward AND NOT #iModeAutoPosCondition AND NOT #iModeSemiAutoPosCondition AND #iNoStopCondition THEN
                           #sCurrent_Step_NB := #S270_UPDATE_NEXT_STEP;
                           #sCheck_Step_Condition := FALSE;
                       END_IF;
                   END_REGION
               #S20_SHUTTLE_TO_STOP_CYCLE_POS_START_REQ:
                   REGION S20_SHUTTLE_TO_STOP_CYCLE_POS_START_REQ
                       IF #sInterface.SequenceReleased AND #sStepForward AND (#iShuttleMoving OR #iShuttleModeAutoPos) THEN
                           #sCurrent_Step_NB := #S30_SHUTTLE_TO_STOP_CYCLE_POS_REACHED;
                           #sCheck_Step_Condition := FALSE;
                       END_IF;
                   END_REGION
               #S30_SHUTTLE_TO_STOP_CYCLE_POS_REACHED:
                   REGION S30_SHUTTLE_TO_STOP_CYCLE_POS_REACHED
                       IF #sInterface.SequenceReleased AND #sStepForward AND NOT #sShuttleStartReq AND #iShuttleModeAutoPos THEN
                           #sCurrent_Step_NB := #S40_STOP_CYCLE;
                           #sCheck_Step_Condition := FALSE;
                       END_IF;
                   END_REGION
               #S40_STOP_CYCLE:
                   REGION S40_STOP_CYCLE
                       IF #sInterface.SequenceReleased AND #sStepForward AND #iNC_Stopped THEN
                           #sCurrent_Step_NB := #S50_WAIT_OPERATOR_RESTART;
                           #sCheck_Step_Condition := FALSE;
                       END_IF;
                   END_REGION
                   #S50_WAIT_OPERATOR_RESTART:
                       REGION S50_WAIT_OPERATOR_RESTART
                           IF #sInterface.SequenceReleased AND #sStepForward AND #iOperatorCycleRestart THEN
                               #sCurrent_Step_NB := #S60_NC_RESTART;
                               #sCheck_Step_Condition := FALSE;
                           END_IF;
                       END_REGION
                   #S60_NC_RESTART:
                       REGION S60_NC_RESTART
                           IF #sInterface.SequenceReleased AND #sStepForward AND #iNC_Running THEN
                               #sCurrent_Step_NB := #S70_UPDATE_NEXT_STEP;
                               #sCheck_Step_Condition := FALSE;
                           END_IF;
                       END_REGION
                   #S70_UPDATE_NEXT_STEP:
                       REGION S70_UPDATE_NEXT_STEP
                           IF #sInterface.SequenceReleased AND #sStepForward AND "AlwaysTRUE" THEN
                               #sCurrent_Step_NB := #S295_JOB_DONE;
                               #sCheck_Step_Condition := FALSE;
                           END_IF;
                       END_REGION

